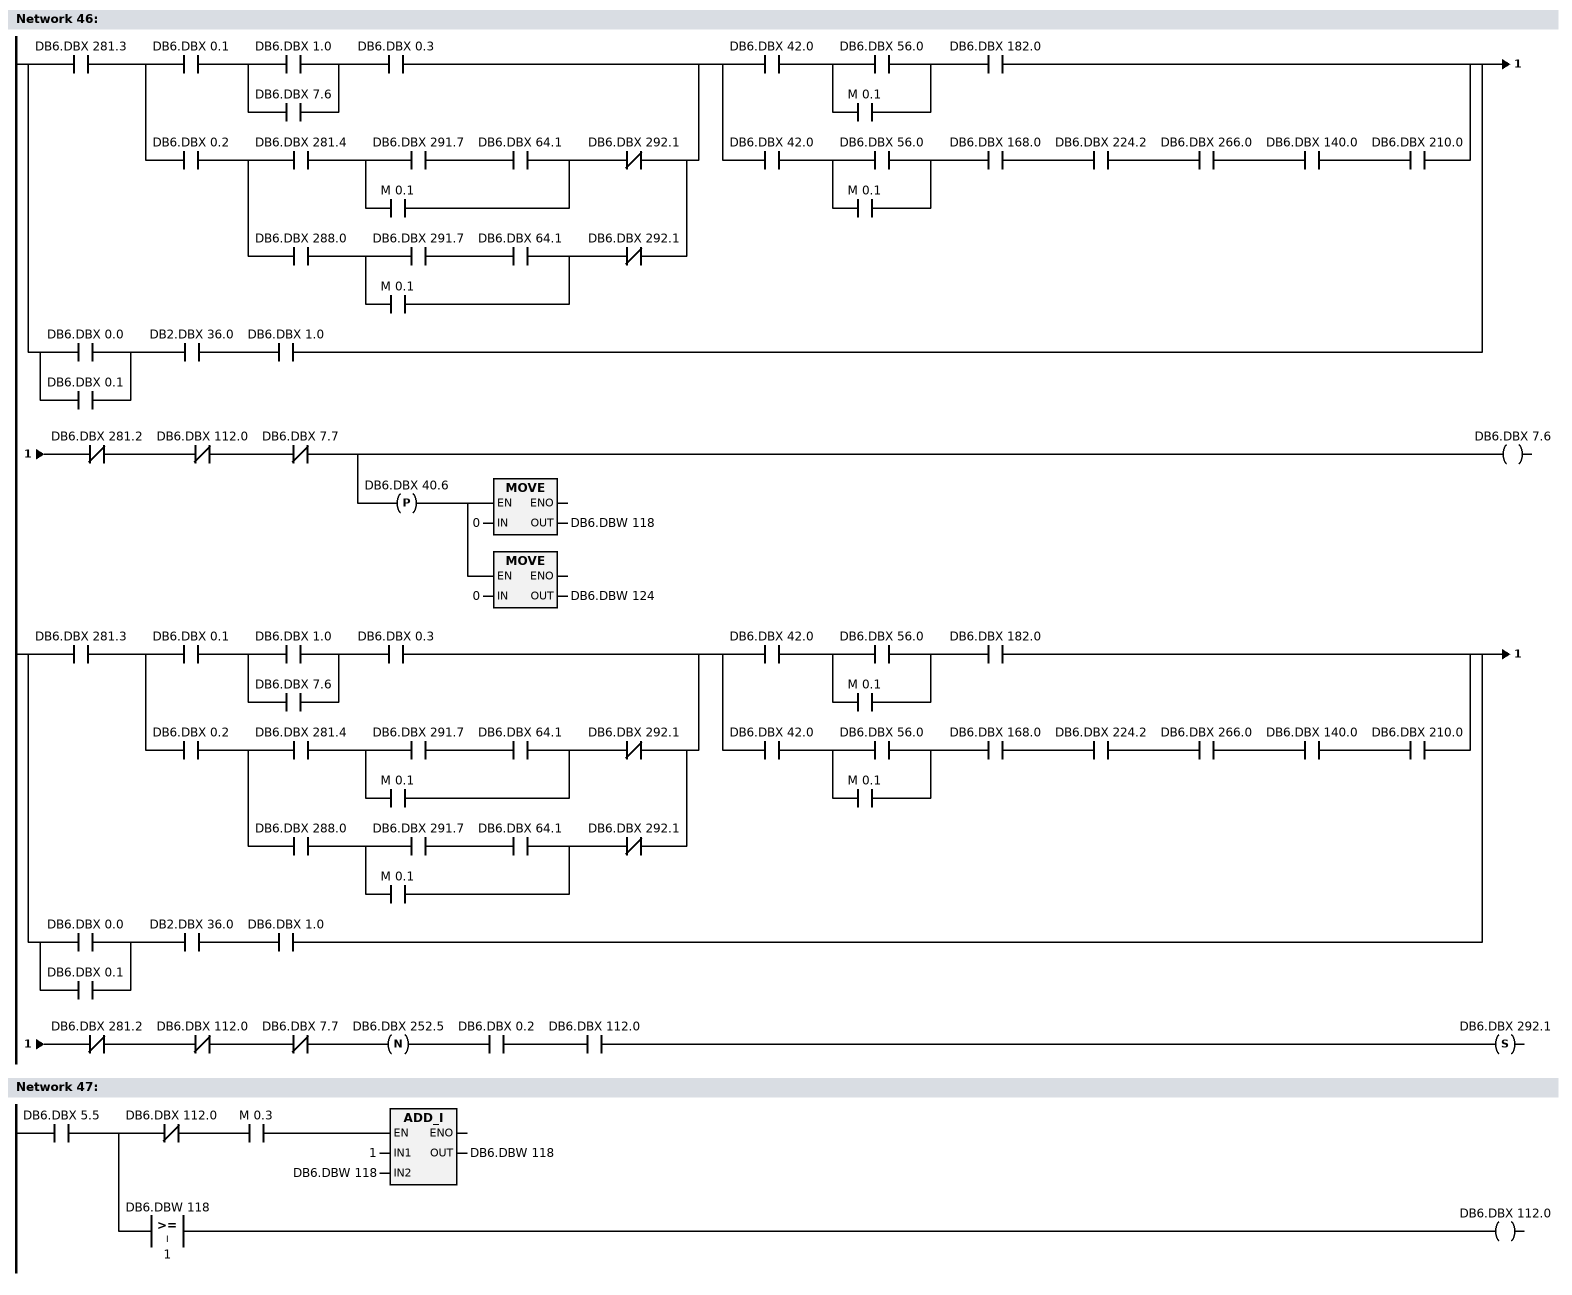
NETWORK
TITLE =
      A(;
      A     DB6.DBX 281.3;
      A(;
      A     DB6.DBX 0.1;
      A(;
      O     DB6.DBX 1.0;
      O     DB6.DBX 7.6;
      );
      A     DB6.DBX 0.3;
      O;
      A     DB6.DBX 0.2;
      A(;
      A     DB6.DBX 281.4;
      A(;
      A     DB6.DBX 291.7;
      A     DB6.DBX 64.1;
      O     M 0.1;
      );
      AN    DB6.DBX 292.1;
      O;
      A     DB6.DBX 288.0;
      A(;
      A     DB6.DBX 291.7;
      A     DB6.DBX 64.1;
      O     M 0.1;
      );
      AN    DB6.DBX 292.1;
      );
      );
      A(;
      A     DB6.DBX 42.0;
      A(;
      O     DB6.DBX 56.0;
      O     M 0.1;
      );
      A     DB6.DBX 182.0;
      O;
      A     DB6.DBX 42.0;
      A(;
      O     DB6.DBX 56.0;
      O     M 0.1;
      );
      A     DB6.DBX 168.0;
      A     DB6.DBX 224.2;
      A     DB6.DBX 266.0;
      A     DB6.DBX 140.0;
      A     DB6.DBX 210.0;
      );
      O;
      A(;
      O     DB6.DBX 0.0;
      O     DB6.DBX 0.1;
      );
      A     DB2.DBX 36.0;
      A     DB6.DBX 1.0;
      );
      AN    DB6.DBX 281.2;
      AN    DB6.DBX 112.0;
      AN    DB6.DBX 7.7;
      =     L 0.0;
      A     L 0.0;
      BLD   102;
      =     DB6.DBX 7.6;
      A(;
      A     L 0.0;
      FN    DB6.DBX 252.5;
      );
      A     DB6.DBX 0.2;
      A     DB6.DBX 112.0;
      S     DB6.DBX 292.1;
      A     L 0.0;
      FP    DB6.DBX 40.6;
      =     L 0.1;
      A     L 0.1;
      JNB   M039;
      L     0;
      T     DB6.DBW 118;
M039: NOP   0;
      A     L 0.1;
      JNB   M040;
      L     0;
      T     DB6.DBW 124;
M040: NOP   0;
NETWORK
TITLE =
      A     DB6.DBX 5.5;
      =     L 0.0;
      A     L 0.0;
      AN    DB6.DBX 112.0;
      A     M 0.3;
      JNB   M041;
      L     1;
      L     DB6.DBW 118;
      +I;
      T     DB6.DBW 118;
M041: NOP   0;
      A     L 0.0;
      A(;
      L     DB6.DBW 118;
      L     1;
      >=I;
      );
      =     DB6.DBX 112.0;
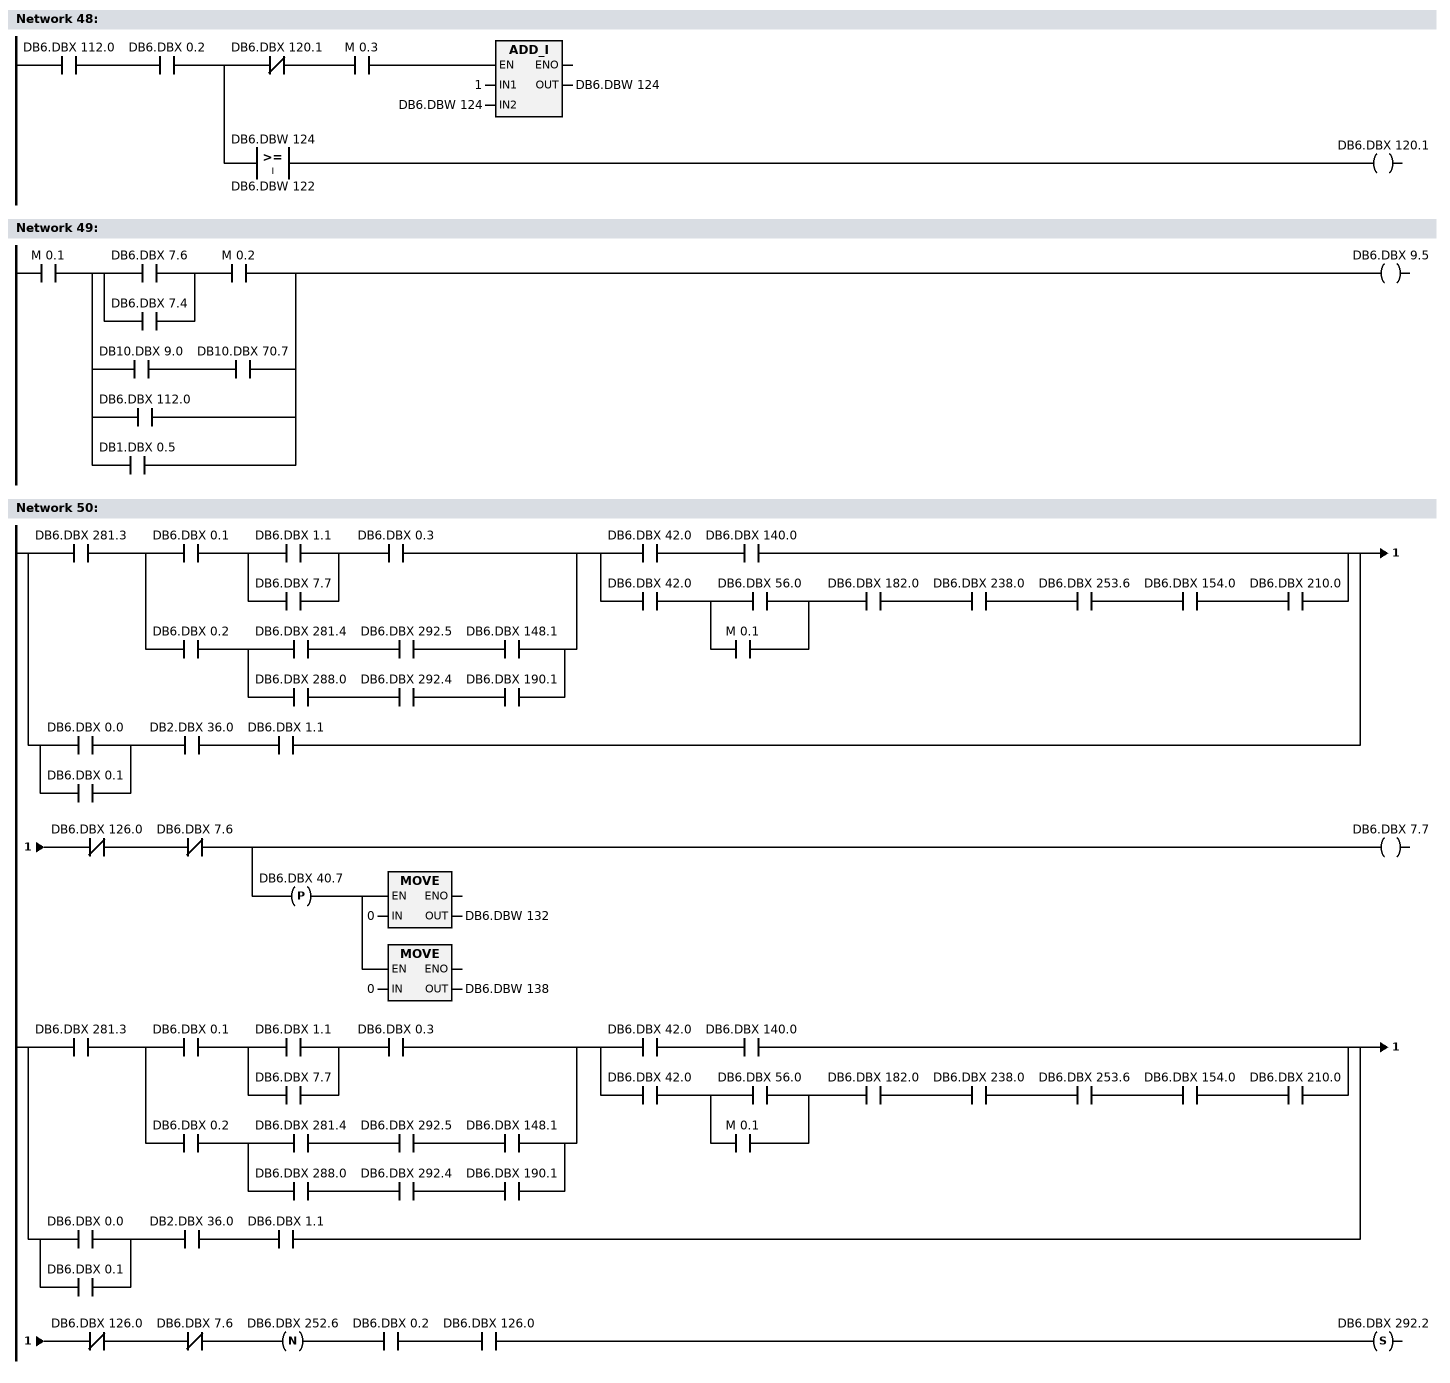
NETWORK
TITLE =
      A     DB6.DBX 112.0;
      A     DB6.DBX 0.2;
      =     L 0.0;
      A     L 0.0;
      AN    DB6.DBX 120.1;
      A     M 0.3;
      JNB   M042;
      L     1;
      L     DB6.DBW 124;
      +I;
      T     DB6.DBW 124;
M042: NOP   0;
      A     L 0.0;
      A(;
      L     DB6.DBW 124;
      L     DB6.DBW 122;
      >=I;
      );
      =     DB6.DBX 120.1;
NETWORK
TITLE =
      A     M 0.1;
      A(;
      A(;
      O     DB6.DBX 7.6;
      O     DB6.DBX 7.4;
      );
      A     M 0.2;
      O;
      A     DB10.DBX 9.0;
      A     DB10.DBX 70.7;
      O     DB6.DBX 112.0;
      O     DB1.DBX 0.5;
      );
      =     DB6.DBX 9.5;
NETWORK
TITLE =
      A(;
      A     DB6.DBX 281.3;
      A(;
      A     DB6.DBX 0.1;
      A(;
      O     DB6.DBX 1.1;
      O     DB6.DBX 7.7;
      );
      A     DB6.DBX 0.3;
      O;
      A     DB6.DBX 0.2;
      A(;
      A     DB6.DBX 281.4;
      A     DB6.DBX 292.5;
      A     DB6.DBX 148.1;
      O;
      A     DB6.DBX 288.0;
      A     DB6.DBX 292.4;
      A     DB6.DBX 190.1;
      );
      );
      A(;
      A     DB6.DBX 42.0;
      A     DB6.DBX 140.0;
      O;
      A     DB6.DBX 42.0;
      A(;
      O     DB6.DBX 56.0;
      O     M 0.1;
      );
      A     DB6.DBX 182.0;
      A     DB6.DBX 238.0;
      A     DB6.DBX 253.6;
      A     DB6.DBX 154.0;
      A     DB6.DBX 210.0;
      );
      O;
      A(;
      O     DB6.DBX 0.0;
      O     DB6.DBX 0.1;
      );
      A     DB2.DBX 36.0;
      A     DB6.DBX 1.1;
      );
      AN    DB6.DBX 126.0;
      AN    DB6.DBX 7.6;
      =     L 0.0;
      A     L 0.0;
      BLD   102;
      =     DB6.DBX 7.7;
      A(;
      A     L 0.0;
      FN    DB6.DBX 252.6;
      );
      A     DB6.DBX 0.2;
      A     DB6.DBX 126.0;
      S     DB6.DBX 292.2;
      A     L 0.0;
      FP    DB6.DBX 40.7;
      =     L 0.1;
      A     L 0.1;
      JNB   M043;
      L     0;
      T     DB6.DBW 132;
M043: NOP   0;
      A     L 0.1;
      JNB   M044;
      L     0;
      T     DB6.DBW 138;
M044: NOP   0;
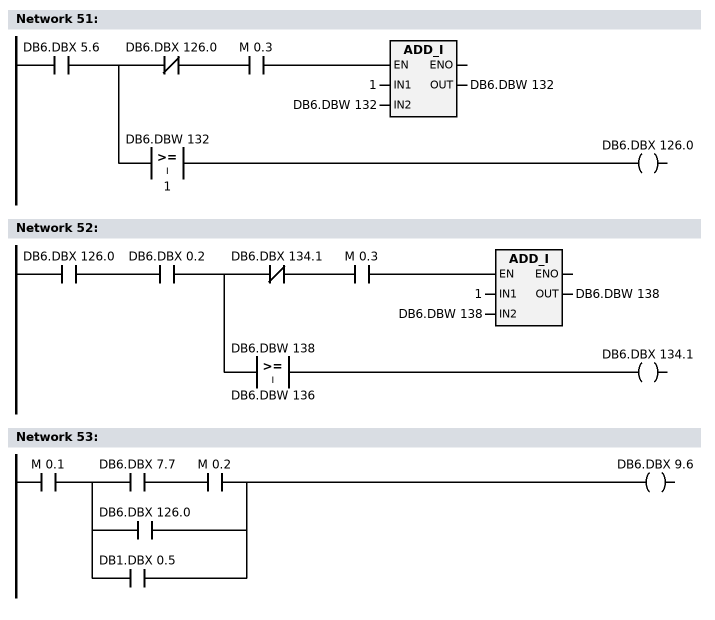
NETWORK
TITLE =
      A     DB6.DBX 5.6;
      =     L 0.0;
      A     L 0.0;
      AN    DB6.DBX 126.0;
      A     M 0.3;
      JNB   M045;
      L     1;
      L     DB6.DBW 132;
      +I;
      T     DB6.DBW 132;
M045: NOP   0;
      A     L 0.0;
      A(;
      L     DB6.DBW 132;
      L     1;
      >=I;
      );
      =     DB6.DBX 126.0;
NETWORK
TITLE =
      A     DB6.DBX 126.0;
      A     DB6.DBX 0.2;
      =     L 0.0;
      A     L 0.0;
      AN    DB6.DBX 134.1;
      A     M 0.3;
      JNB   M046;
      L     1;
      L     DB6.DBW 138;
      +I;
      T     DB6.DBW 138;
M046: NOP   0;
      A     L 0.0;
      A(;
      L     DB6.DBW 138;
      L     DB6.DBW 136;
      >=I;
      );
      =     DB6.DBX 134.1;
NETWORK
TITLE =
      A     M 0.1;
      A(;
      A     DB6.DBX 7.7;
      A     M 0.2;
      O     DB6.DBX 126.0;
      O     DB1.DBX 0.5;
      );
      =     DB6.DBX 9.6;
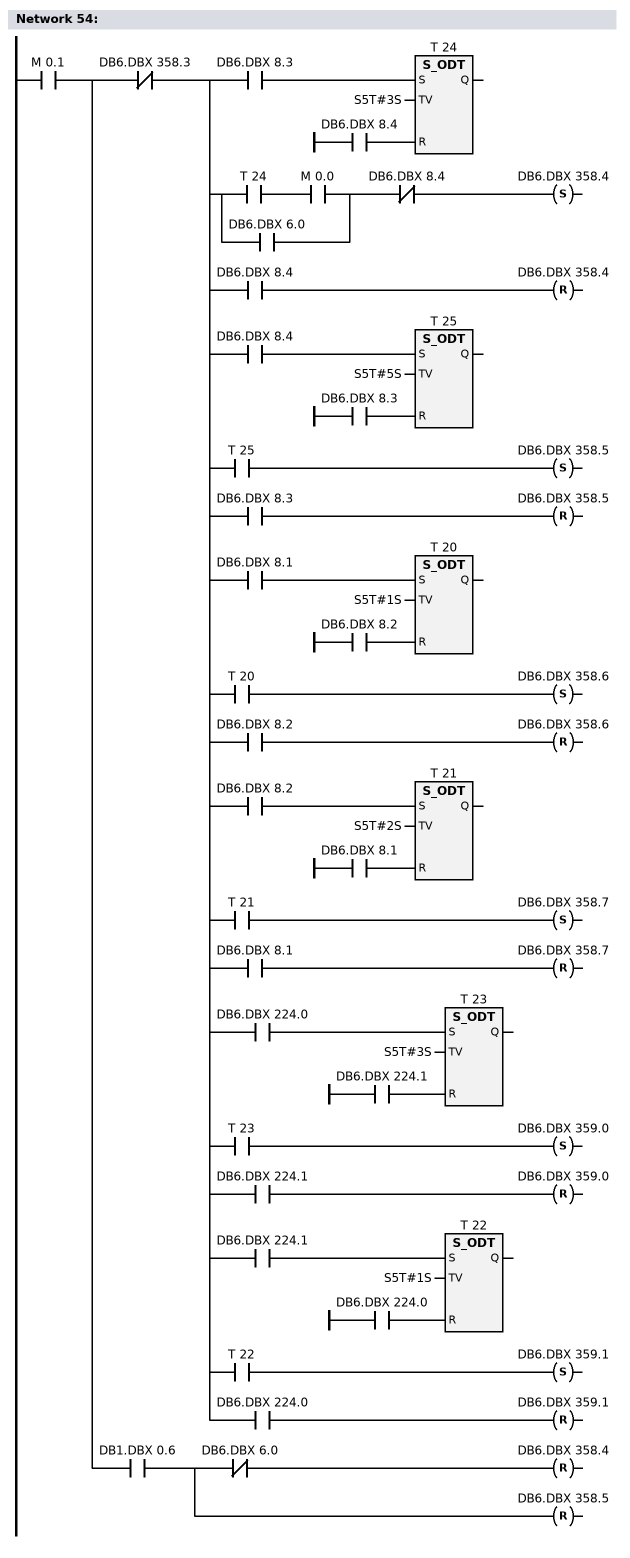
NETWORK
TITLE =
      A     M 0.1;
      =     L 0.0;
      A     L 0.0;
      AN    DB6.DBX 358.3;
      =     L 0.1;
      A     L 0.1;
      A     DB6.DBX 8.3;
      L     S5T#3S;
      SD    T 24;
      A     DB6.DBX 8.4;
      R     T 24;
      NOP   0;
      NOP   0;
      NOP   0;
      A     L 0.1;
      A(;
      A     T 24;
      A     M 0.0;
      O     DB6.DBX 6.0;
      );
      AN    DB6.DBX 8.4;
      S     DB6.DBX 358.4;
      A     L 0.1;
      A     DB6.DBX 8.4;
      R     DB6.DBX 358.4;
      A     L 0.1;
      A     DB6.DBX 8.4;
      L     S5T#5S;
      SD    T 25;
      A     DB6.DBX 8.3;
      R     T 25;
      NOP   0;
      NOP   0;
      NOP   0;
      A     L 0.1;
      A     T 25;
      S     DB6.DBX 358.5;
      A     L 0.1;
      A     DB6.DBX 8.3;
      R     DB6.DBX 358.5;
      A     L 0.1;
      A     DB6.DBX 8.1;
      L     S5T#1S;
      SD    T 20;
      A     DB6.DBX 8.2;
      R     T 20;
      NOP   0;
      NOP   0;
      NOP   0;
      A     L 0.1;
      A     T 20;
      S     DB6.DBX 358.6;
      A     L 0.1;
      A     DB6.DBX 8.2;
      R     DB6.DBX 358.6;
      A     L 0.1;
      A     DB6.DBX 8.2;
      L     S5T#2S;
      SD    T 21;
      A     DB6.DBX 8.1;
      R     T 21;
      NOP   0;
      NOP   0;
      NOP   0;
      A     L 0.1;
      A     T 21;
      S     DB6.DBX 358.7;
      A     L 0.1;
      A     DB6.DBX 8.1;
      R     DB6.DBX 358.7;
      A     L 0.1;
      A     DB6.DBX 224.0;
      L     S5T#3S;
      SD    T 23;
      A     DB6.DBX 224.1;
      R     T 23;
      NOP   0;
      NOP   0;
      NOP   0;
      A     L 0.1;
      A     T 23;
      S     DB6.DBX 359.0;
      A     L 0.1;
      A     DB6.DBX 224.1;
      R     DB6.DBX 359.0;
      A     L 0.1;
      A     DB6.DBX 224.1;
      L     S5T#1S;
      SD    T 22;
      A     DB6.DBX 224.0;
      R     T 22;
      NOP   0;
      NOP   0;
      NOP   0;
      A     L 0.1;
      A     T 22;
      S     DB6.DBX 359.1;
      A     L 0.1;
      A     DB6.DBX 224.0;
      R     DB6.DBX 359.1;
      A     L 0.0;
      A     DB1.DBX 0.6;
      =     L 0.1;
      A     L 0.1;
      AN    DB6.DBX 6.0;
      R     DB6.DBX 358.4;
      A     L 0.1;
      BLD   102;
      R     DB6.DBX 358.5;
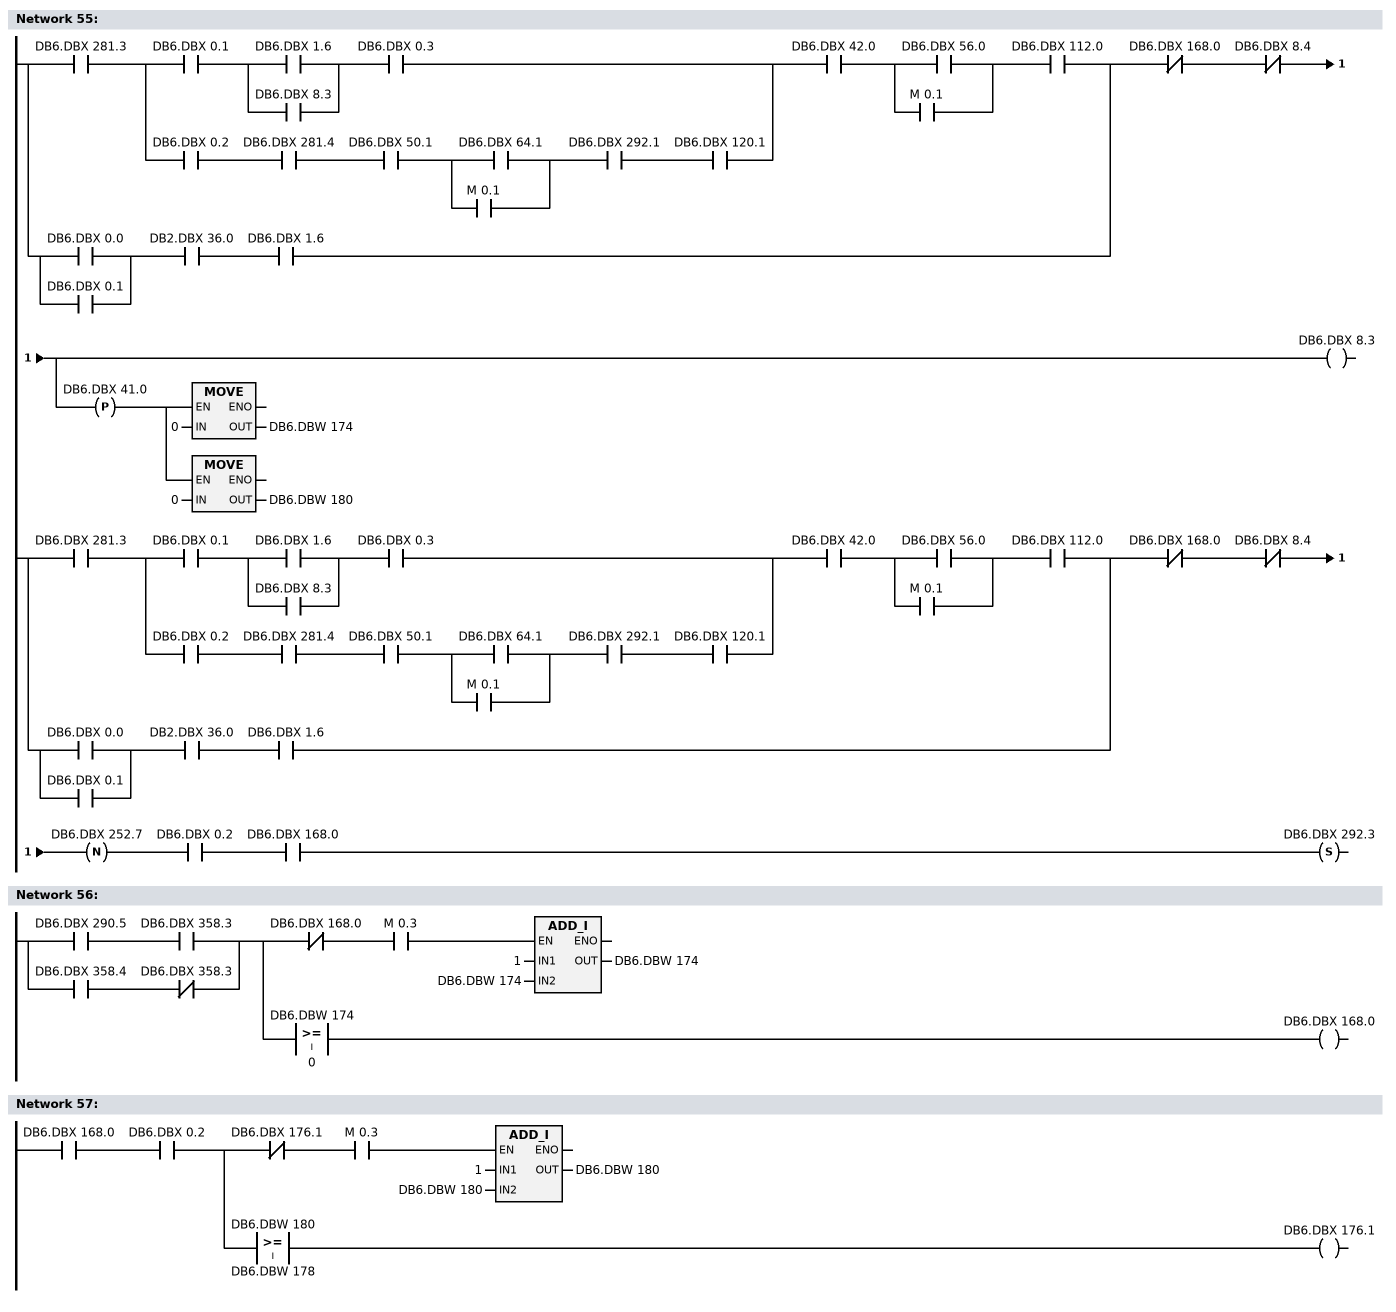
NETWORK
TITLE =
      A(;
      A     DB6.DBX 281.3;
      A(;
      A     DB6.DBX 0.1;
      A(;
      O     DB6.DBX 1.6;
      O     DB6.DBX 8.3;
      );
      A     DB6.DBX 0.3;
      O;
      A     DB6.DBX 0.2;
      A     DB6.DBX 281.4;
      A     DB6.DBX 50.1;
      A(;
      O     DB6.DBX 64.1;
      O     M 0.1;
      );
      A     DB6.DBX 292.1;
      A     DB6.DBX 120.1;
      );
      A     DB6.DBX 42.0;
      A(;
      O     DB6.DBX 56.0;
      O     M 0.1;
      );
      A     DB6.DBX 112.0;
      O;
      A(;
      O     DB6.DBX 0.0;
      O     DB6.DBX 0.1;
      );
      A     DB2.DBX 36.0;
      A     DB6.DBX 1.6;
      );
      AN    DB6.DBX 168.0;
      AN    DB6.DBX 8.4;
      =     L 0.0;
      A     L 0.0;
      BLD   102;
      =     DB6.DBX 8.3;
      A(;
      A     L 0.0;
      FN    DB6.DBX 252.7;
      );
      A     DB6.DBX 0.2;
      A     DB6.DBX 168.0;
      S     DB6.DBX 292.3;
      A     L 0.0;
      FP    DB6.DBX 41.0;
      =     L 0.1;
      A     L 0.1;
      JNB   M047;
      L     0;
      T     DB6.DBW 174;
M047: NOP   0;
      A     L 0.1;
      JNB   M048;
      L     0;
      T     DB6.DBW 180;
M048: NOP   0;
NETWORK
TITLE =
      A     DB6.DBX 290.5;
      A     DB6.DBX 358.3;
      O;
      A     DB6.DBX 358.4;
      AN    DB6.DBX 358.3;
      =     L 0.0;
      A     L 0.0;
      AN    DB6.DBX 168.0;
      A     M 0.3;
      JNB   M049;
      L     1;
      L     DB6.DBW 174;
      +I;
      T     DB6.DBW 174;
M049: NOP   0;
      A     L 0.0;
      A(;
      L     DB6.DBW 174;
      L     0;
      >=I;
      );
      =     DB6.DBX 168.0;
NETWORK
TITLE =
      A     DB6.DBX 168.0;
      A     DB6.DBX 0.2;
      =     L 0.0;
      A     L 0.0;
      AN    DB6.DBX 176.1;
      A     M 0.3;
      JNB   M050;
      L     1;
      L     DB6.DBW 180;
      +I;
      T     DB6.DBW 180;
M050: NOP   0;
      A     L 0.0;
      A(;
      L     DB6.DBW 180;
      L     DB6.DBW 178;
      >=I;
      );
      =     DB6.DBX 176.1;
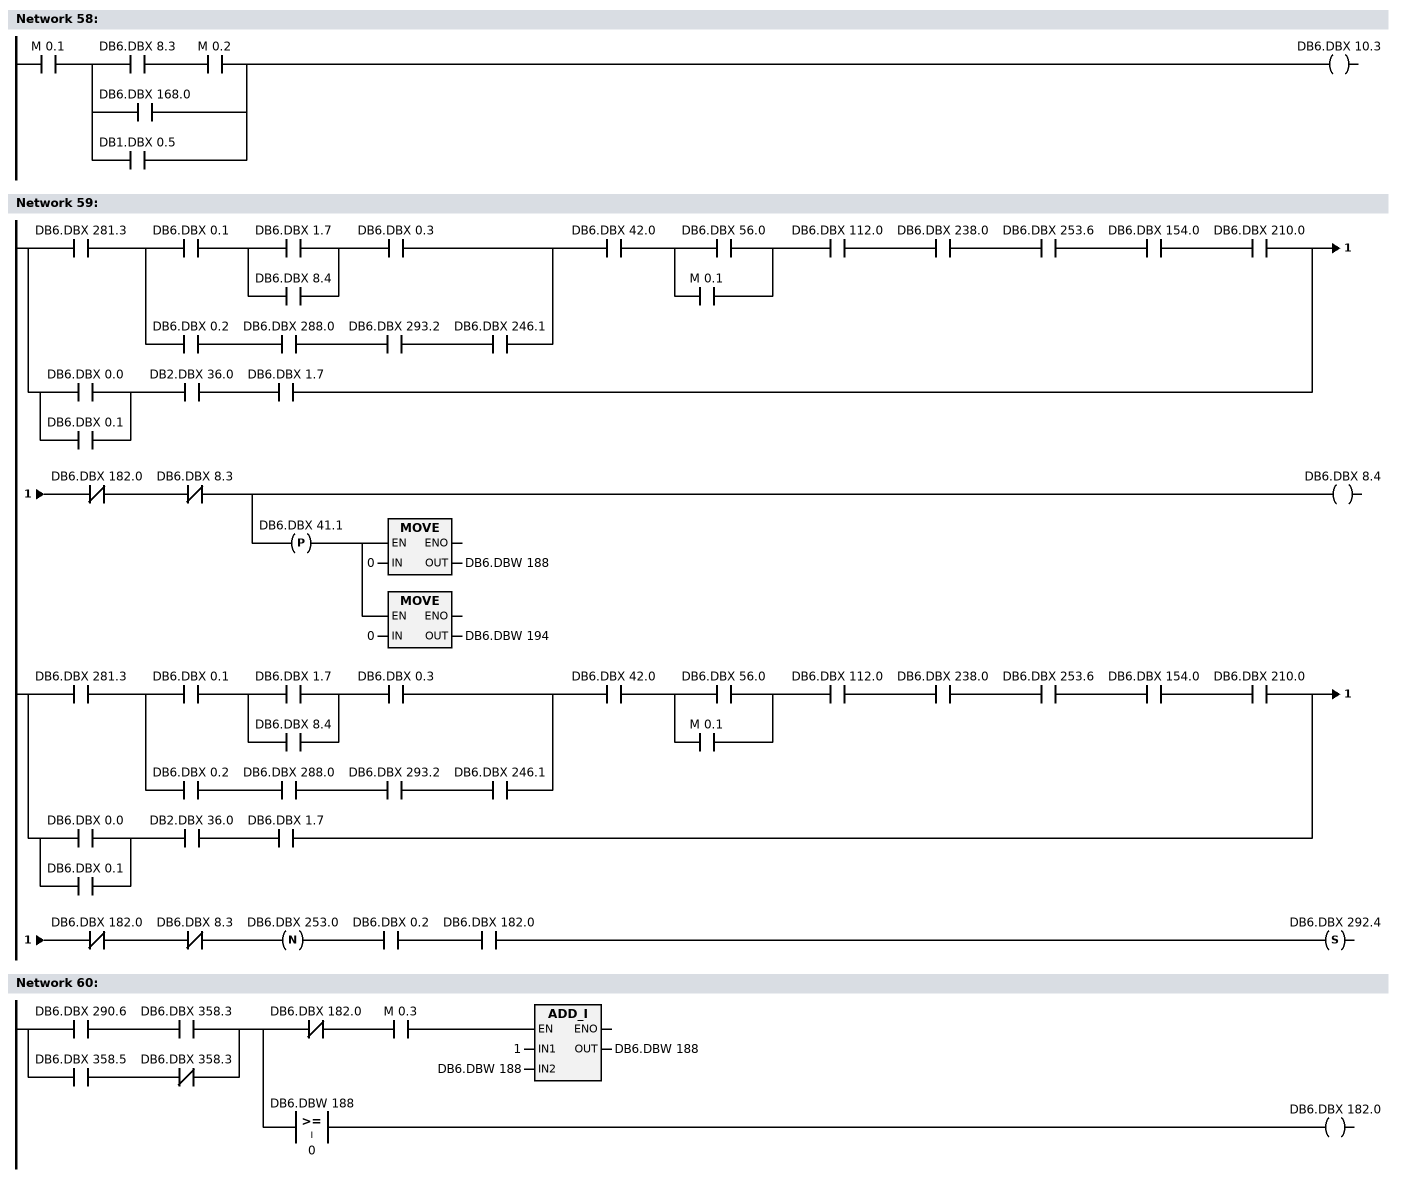
NETWORK
TITLE =
      A     M 0.1;
      A(;
      A     DB6.DBX 8.3;
      A     M 0.2;
      O     DB6.DBX 168.0;
      O     DB1.DBX 0.5;
      );
      =     DB6.DBX 10.3;
NETWORK
TITLE =
      A(;
      A     DB6.DBX 281.3;
      A(;
      A     DB6.DBX 0.1;
      A(;
      O     DB6.DBX 1.7;
      O     DB6.DBX 8.4;
      );
      A     DB6.DBX 0.3;
      O;
      A     DB6.DBX 0.2;
      A     DB6.DBX 288.0;
      A     DB6.DBX 293.2;
      A     DB6.DBX 246.1;
      );
      A     DB6.DBX 42.0;
      A(;
      O     DB6.DBX 56.0;
      O     M 0.1;
      );
      A     DB6.DBX 112.0;
      A     DB6.DBX 238.0;
      A     DB6.DBX 253.6;
      A     DB6.DBX 154.0;
      A     DB6.DBX 210.0;
      O;
      A(;
      O     DB6.DBX 0.0;
      O     DB6.DBX 0.1;
      );
      A     DB2.DBX 36.0;
      A     DB6.DBX 1.7;
      );
      AN    DB6.DBX 182.0;
      AN    DB6.DBX 8.3;
      =     L 0.0;
      A     L 0.0;
      BLD   102;
      =     DB6.DBX 8.4;
      A(;
      A     L 0.0;
      FN    DB6.DBX 253.0;
      );
      A     DB6.DBX 0.2;
      A     DB6.DBX 182.0;
      S     DB6.DBX 292.4;
      A     L 0.0;
      FP    DB6.DBX 41.1;
      =     L 0.1;
      A     L 0.1;
      JNB   M051;
      L     0;
      T     DB6.DBW 188;
M051: NOP   0;
      A     L 0.1;
      JNB   M052;
      L     0;
      T     DB6.DBW 194;
M052: NOP   0;
NETWORK
TITLE =
      A     DB6.DBX 290.6;
      A     DB6.DBX 358.3;
      O;
      A     DB6.DBX 358.5;
      AN    DB6.DBX 358.3;
      =     L 0.0;
      A     L 0.0;
      AN    DB6.DBX 182.0;
      A     M 0.3;
      JNB   M053;
      L     1;
      L     DB6.DBW 188;
      +I;
      T     DB6.DBW 188;
M053: NOP   0;
      A     L 0.0;
      A(;
      L     DB6.DBW 188;
      L     0;
      >=I;
      );
      =     DB6.DBX 182.0;
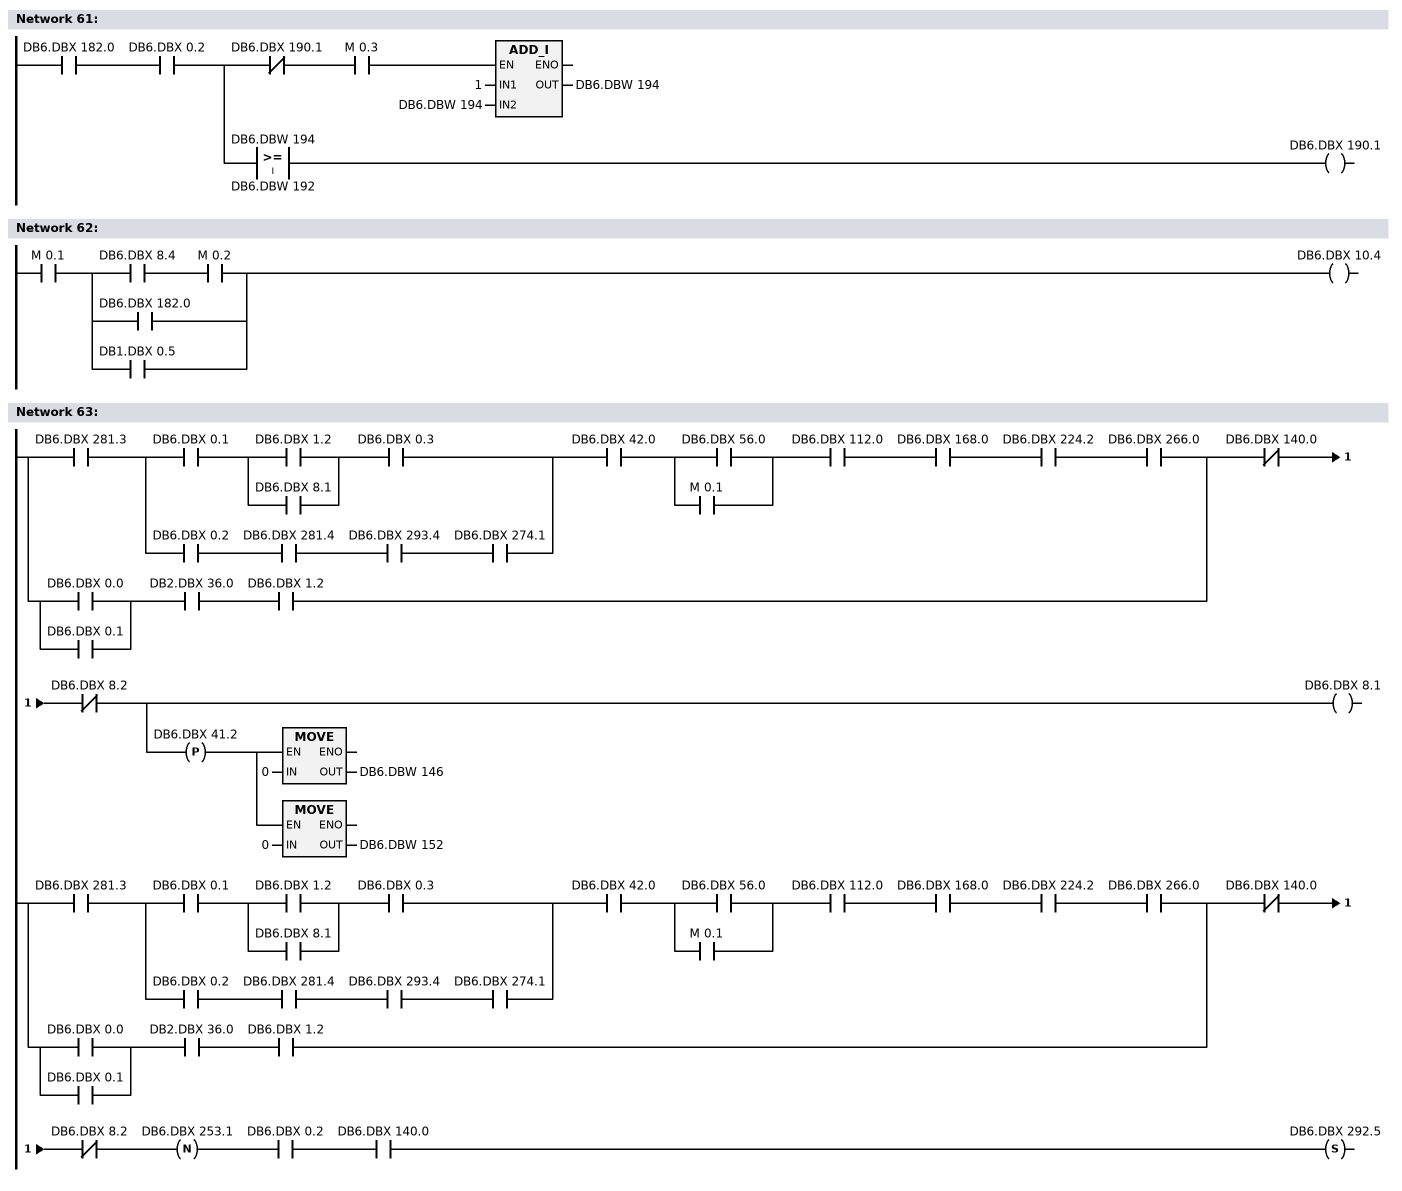
NETWORK
TITLE =
      A     DB6.DBX 182.0;
      A     DB6.DBX 0.2;
      =     L 0.0;
      A     L 0.0;
      AN    DB6.DBX 190.1;
      A     M 0.3;
      JNB   M054;
      L     1;
      L     DB6.DBW 194;
      +I;
      T     DB6.DBW 194;
M054: NOP   0;
      A     L 0.0;
      A(;
      L     DB6.DBW 194;
      L     DB6.DBW 192;
      >=I;
      );
      =     DB6.DBX 190.1;
NETWORK
TITLE =
      A     M 0.1;
      A(;
      A     DB6.DBX 8.4;
      A     M 0.2;
      O     DB6.DBX 182.0;
      O     DB1.DBX 0.5;
      );
      =     DB6.DBX 10.4;
NETWORK
TITLE =
      A(;
      A     DB6.DBX 281.3;
      A(;
      A     DB6.DBX 0.1;
      A(;
      O     DB6.DBX 1.2;
      O     DB6.DBX 8.1;
      );
      A     DB6.DBX 0.3;
      O;
      A     DB6.DBX 0.2;
      A     DB6.DBX 281.4;
      A     DB6.DBX 293.4;
      A     DB6.DBX 274.1;
      );
      A     DB6.DBX 42.0;
      A(;
      O     DB6.DBX 56.0;
      O     M 0.1;
      );
      A     DB6.DBX 112.0;
      A     DB6.DBX 168.0;
      A     DB6.DBX 224.2;
      A     DB6.DBX 266.0;
      O;
      A(;
      O     DB6.DBX 0.0;
      O     DB6.DBX 0.1;
      );
      A     DB2.DBX 36.0;
      A     DB6.DBX 1.2;
      );
      AN    DB6.DBX 140.0;
      AN    DB6.DBX 8.2;
      =     L 0.0;
      A     L 0.0;
      BLD   102;
      =     DB6.DBX 8.1;
      A(;
      A     L 0.0;
      FN    DB6.DBX 253.1;
      );
      A     DB6.DBX 0.2;
      A     DB6.DBX 140.0;
      S     DB6.DBX 292.5;
      A     L 0.0;
      FP    DB6.DBX 41.2;
      =     L 0.1;
      A     L 0.1;
      JNB   M055;
      L     0;
      T     DB6.DBW 146;
M055: NOP   0;
      A     L 0.1;
      JNB   M056;
      L     0;
      T     DB6.DBW 152;
M056: NOP   0;
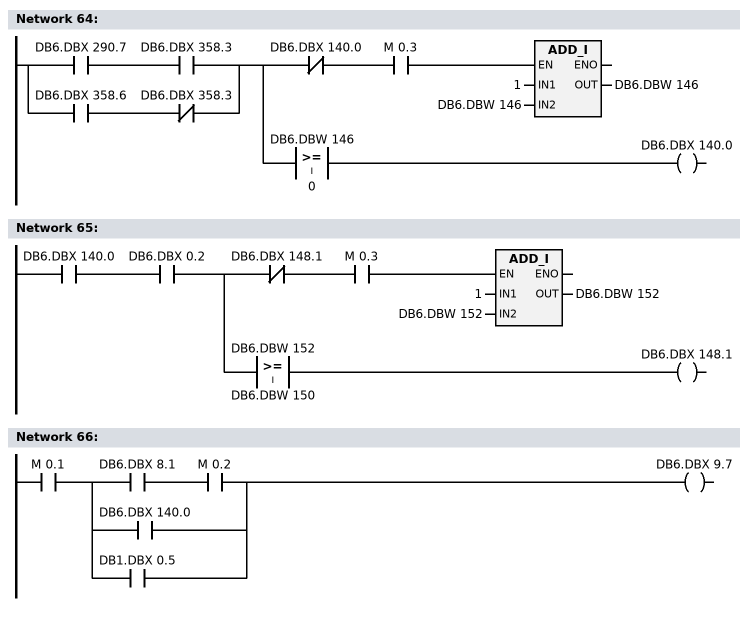
NETWORK
TITLE =
      A     DB6.DBX 290.7;
      A     DB6.DBX 358.3;
      O;
      A     DB6.DBX 358.6;
      AN    DB6.DBX 358.3;
      =     L 0.0;
      A     L 0.0;
      AN    DB6.DBX 140.0;
      A     M 0.3;
      JNB   M057;
      L     1;
      L     DB6.DBW 146;
      +I;
      T     DB6.DBW 146;
M057: NOP   0;
      A     L 0.0;
      A(;
      L     DB6.DBW 146;
      L     0;
      >=I;
      );
      =     DB6.DBX 140.0;
NETWORK
TITLE =
      A     DB6.DBX 140.0;
      A     DB6.DBX 0.2;
      =     L 0.0;
      A     L 0.0;
      AN    DB6.DBX 148.1;
      A     M 0.3;
      JNB   M058;
      L     1;
      L     DB6.DBW 152;
      +I;
      T     DB6.DBW 152;
M058: NOP   0;
      A     L 0.0;
      A(;
      L     DB6.DBW 152;
      L     DB6.DBW 150;
      >=I;
      );
      =     DB6.DBX 148.1;
NETWORK
TITLE =
      A     M 0.1;
      A(;
      A     DB6.DBX 8.1;
      A     M 0.2;
      O     DB6.DBX 140.0;
      O     DB1.DBX 0.5;
      );
      =     DB6.DBX 9.7;
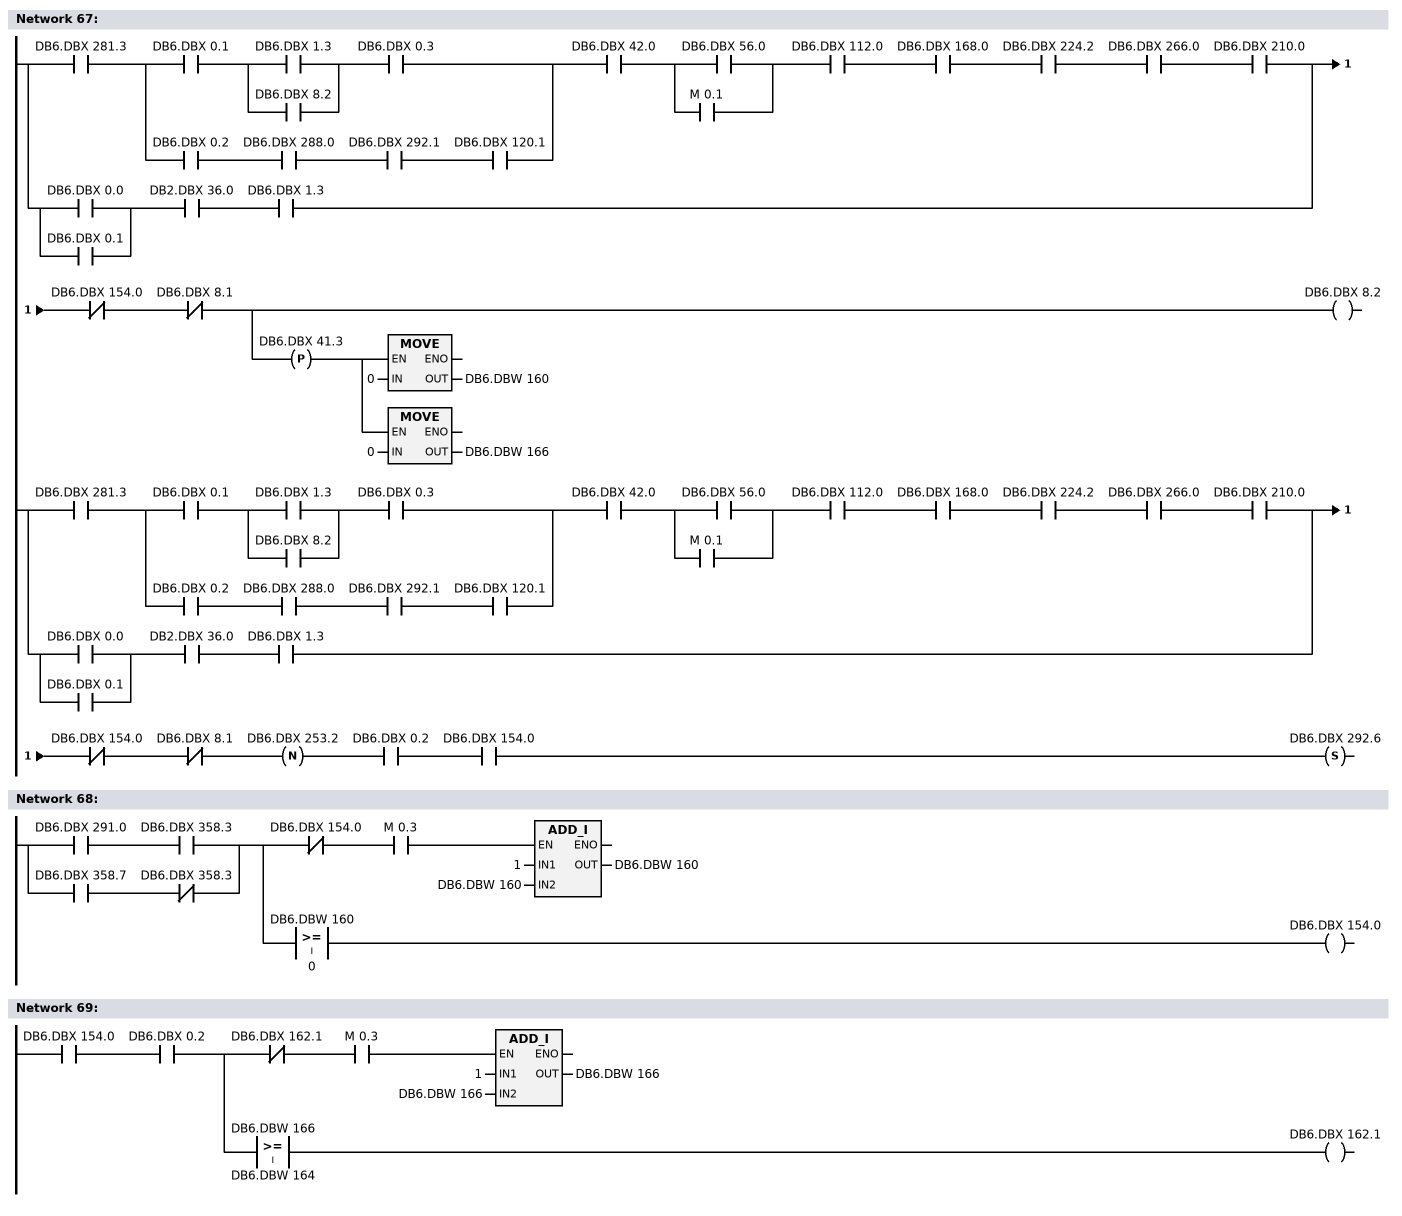
NETWORK
TITLE =
      A(;
      A     DB6.DBX 281.3;
      A(;
      A     DB6.DBX 0.1;
      A(;
      O     DB6.DBX 1.3;
      O     DB6.DBX 8.2;
      );
      A     DB6.DBX 0.3;
      O;
      A     DB6.DBX 0.2;
      A     DB6.DBX 288.0;
      A     DB6.DBX 292.1;
      A     DB6.DBX 120.1;
      );
      A     DB6.DBX 42.0;
      A(;
      O     DB6.DBX 56.0;
      O     M 0.1;
      );
      A     DB6.DBX 112.0;
      A     DB6.DBX 168.0;
      A     DB6.DBX 224.2;
      A     DB6.DBX 266.0;
      A     DB6.DBX 210.0;
      O;
      A(;
      O     DB6.DBX 0.0;
      O     DB6.DBX 0.1;
      );
      A     DB2.DBX 36.0;
      A     DB6.DBX 1.3;
      );
      AN    DB6.DBX 154.0;
      AN    DB6.DBX 8.1;
      =     L 0.0;
      A     L 0.0;
      BLD   102;
      =     DB6.DBX 8.2;
      A(;
      A     L 0.0;
      FN    DB6.DBX 253.2;
      );
      A     DB6.DBX 0.2;
      A     DB6.DBX 154.0;
      S     DB6.DBX 292.6;
      A     L 0.0;
      FP    DB6.DBX 41.3;
      =     L 0.1;
      A     L 0.1;
      JNB   M059;
      L     0;
      T     DB6.DBW 160;
M059: NOP   0;
      A     L 0.1;
      JNB   M060;
      L     0;
      T     DB6.DBW 166;
M060: NOP   0;
NETWORK
TITLE =
      A     DB6.DBX 291.0;
      A     DB6.DBX 358.3;
      O;
      A     DB6.DBX 358.7;
      AN    DB6.DBX 358.3;
      =     L 0.0;
      A     L 0.0;
      AN    DB6.DBX 154.0;
      A     M 0.3;
      JNB   M061;
      L     1;
      L     DB6.DBW 160;
      +I;
      T     DB6.DBW 160;
M061: NOP   0;
      A     L 0.0;
      A(;
      L     DB6.DBW 160;
      L     0;
      >=I;
      );
      =     DB6.DBX 154.0;
NETWORK
TITLE =
      A     DB6.DBX 154.0;
      A     DB6.DBX 0.2;
      =     L 0.0;
      A     L 0.0;
      AN    DB6.DBX 162.1;
      A     M 0.3;
      JNB   M062;
      L     1;
      L     DB6.DBW 166;
      +I;
      T     DB6.DBW 166;
M062: NOP   0;
      A     L 0.0;
      A(;
      L     DB6.DBW 166;
      L     DB6.DBW 164;
      >=I;
      );
      =     DB6.DBX 162.1;
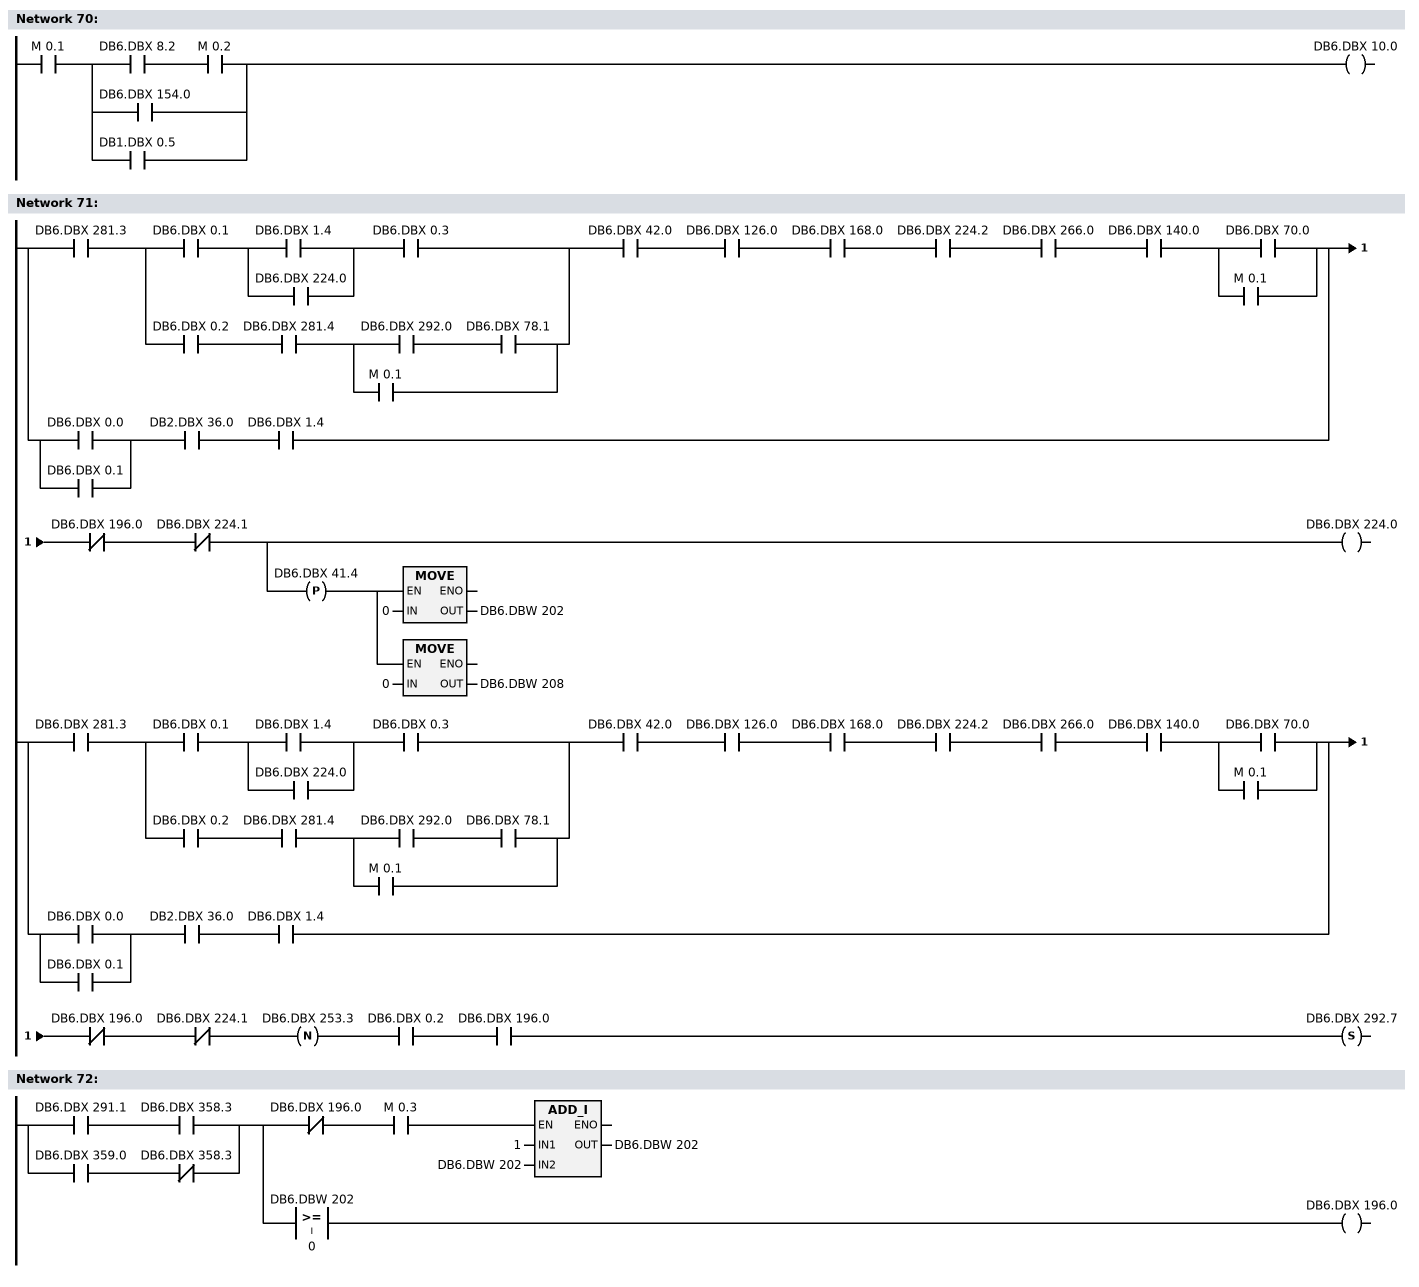
NETWORK
TITLE =
      A     M 0.1;
      A(;
      A     DB6.DBX 8.2;
      A     M 0.2;
      O     DB6.DBX 154.0;
      O     DB1.DBX 0.5;
      );
      =     DB6.DBX 10.0;
NETWORK
TITLE =
      A(;
      A     DB6.DBX 281.3;
      A(;
      A     DB6.DBX 0.1;
      A(;
      O     DB6.DBX 1.4;
      O     DB6.DBX 224.0;
      );
      A     DB6.DBX 0.3;
      O;
      A     DB6.DBX 0.2;
      A     DB6.DBX 281.4;
      A(;
      A     DB6.DBX 292.0;
      A     DB6.DBX 78.1;
      O     M 0.1;
      );
      );
      A     DB6.DBX 42.0;
      A     DB6.DBX 126.0;
      A     DB6.DBX 168.0;
      A     DB6.DBX 224.2;
      A     DB6.DBX 266.0;
      A     DB6.DBX 140.0;
      A(;
      O     DB6.DBX 70.0;
      O     M 0.1;
      );
      O;
      A(;
      O     DB6.DBX 0.0;
      O     DB6.DBX 0.1;
      );
      A     DB2.DBX 36.0;
      A     DB6.DBX 1.4;
      );
      AN    DB6.DBX 196.0;
      AN    DB6.DBX 224.1;
      =     L 0.0;
      A     L 0.0;
      BLD   102;
      =     DB6.DBX 224.0;
      A(;
      A     L 0.0;
      FN    DB6.DBX 253.3;
      );
      A     DB6.DBX 0.2;
      A     DB6.DBX 196.0;
      S     DB6.DBX 292.7;
      A     L 0.0;
      FP    DB6.DBX 41.4;
      =     L 0.1;
      A     L 0.1;
      JNB   M063;
      L     0;
      T     DB6.DBW 202;
M063: NOP   0;
      A     L 0.1;
      JNB   M064;
      L     0;
      T     DB6.DBW 208;
M064: NOP   0;
NETWORK
TITLE =
      A     DB6.DBX 291.1;
      A     DB6.DBX 358.3;
      O;
      A     DB6.DBX 359.0;
      AN    DB6.DBX 358.3;
      =     L 0.0;
      A     L 0.0;
      AN    DB6.DBX 196.0;
      A     M 0.3;
      JNB   M065;
      L     1;
      L     DB6.DBW 202;
      +I;
      T     DB6.DBW 202;
M065: NOP   0;
      A     L 0.0;
      A(;
      L     DB6.DBW 202;
      L     0;
      >=I;
      );
      =     DB6.DBX 196.0;
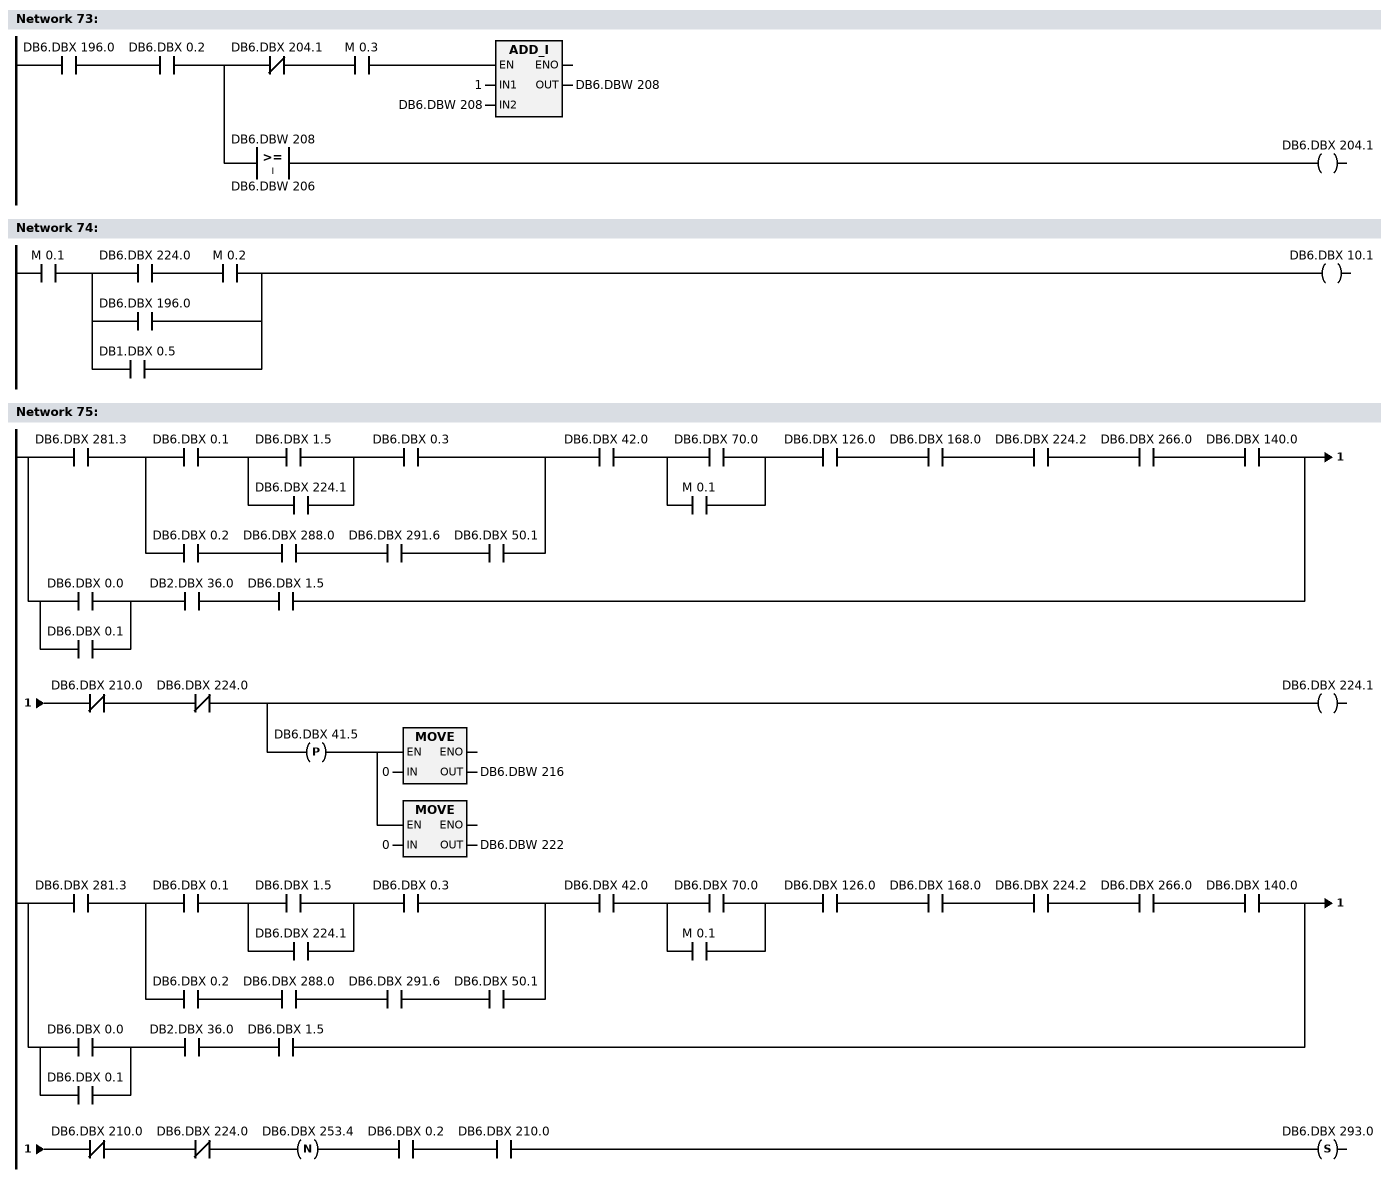
NETWORK
TITLE =
      A     DB6.DBX 196.0;
      A     DB6.DBX 0.2;
      =     L 0.0;
      A     L 0.0;
      AN    DB6.DBX 204.1;
      A     M 0.3;
      JNB   M066;
      L     1;
      L     DB6.DBW 208;
      +I;
      T     DB6.DBW 208;
M066: NOP   0;
      A     L 0.0;
      A(;
      L     DB6.DBW 208;
      L     DB6.DBW 206;
      >=I;
      );
      =     DB6.DBX 204.1;
NETWORK
TITLE =
      A     M 0.1;
      A(;
      A     DB6.DBX 224.0;
      A     M 0.2;
      O     DB6.DBX 196.0;
      O     DB1.DBX 0.5;
      );
      =     DB6.DBX 10.1;
NETWORK
TITLE =
      A(;
      A     DB6.DBX 281.3;
      A(;
      A     DB6.DBX 0.1;
      A(;
      O     DB6.DBX 1.5;
      O     DB6.DBX 224.1;
      );
      A     DB6.DBX 0.3;
      O;
      A     DB6.DBX 0.2;
      A     DB6.DBX 288.0;
      A     DB6.DBX 291.6;
      A     DB6.DBX 50.1;
      );
      A     DB6.DBX 42.0;
      A(;
      O     DB6.DBX 70.0;
      O     M 0.1;
      );
      A     DB6.DBX 126.0;
      A     DB6.DBX 168.0;
      A     DB6.DBX 224.2;
      A     DB6.DBX 266.0;
      A     DB6.DBX 140.0;
      O;
      A(;
      O     DB6.DBX 0.0;
      O     DB6.DBX 0.1;
      );
      A     DB2.DBX 36.0;
      A     DB6.DBX 1.5;
      );
      AN    DB6.DBX 210.0;
      AN    DB6.DBX 224.0;
      =     L 0.0;
      A     L 0.0;
      BLD   102;
      =     DB6.DBX 224.1;
      A(;
      A     L 0.0;
      FN    DB6.DBX 253.4;
      );
      A     DB6.DBX 0.2;
      A     DB6.DBX 210.0;
      S     DB6.DBX 293.0;
      A     L 0.0;
      FP    DB6.DBX 41.5;
      =     L 0.1;
      A     L 0.1;
      JNB   M067;
      L     0;
      T     DB6.DBW 216;
M067: NOP   0;
      A     L 0.1;
      JNB   M068;
      L     0;
      T     DB6.DBW 222;
M068: NOP   0;
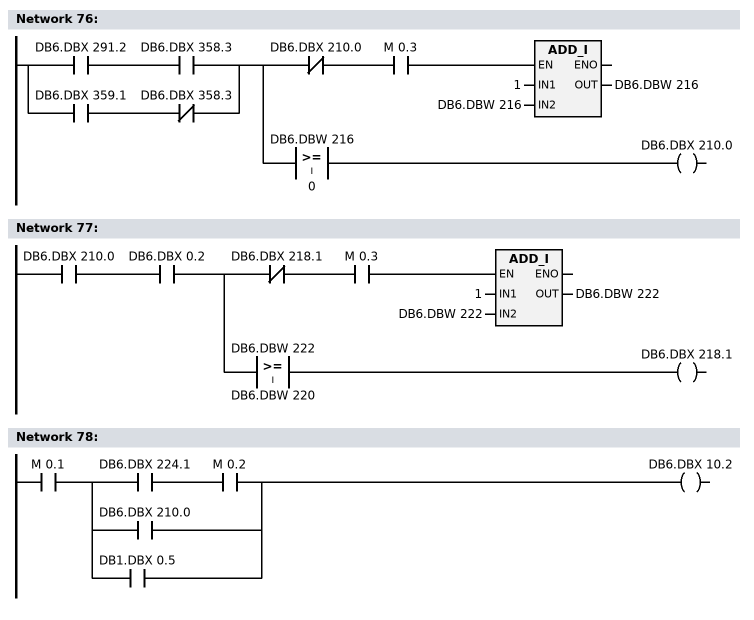
NETWORK
TITLE =
      A     DB6.DBX 291.2;
      A     DB6.DBX 358.3;
      O;
      A     DB6.DBX 359.1;
      AN    DB6.DBX 358.3;
      =     L 0.0;
      A     L 0.0;
      AN    DB6.DBX 210.0;
      A     M 0.3;
      JNB   M069;
      L     1;
      L     DB6.DBW 216;
      +I;
      T     DB6.DBW 216;
M069: NOP   0;
      A     L 0.0;
      A(;
      L     DB6.DBW 216;
      L     0;
      >=I;
      );
      =     DB6.DBX 210.0;
NETWORK
TITLE =
      A     DB6.DBX 210.0;
      A     DB6.DBX 0.2;
      =     L 0.0;
      A     L 0.0;
      AN    DB6.DBX 218.1;
      A     M 0.3;
      JNB   M070;
      L     1;
      L     DB6.DBW 222;
      +I;
      T     DB6.DBW 222;
M070: NOP   0;
      A     L 0.0;
      A(;
      L     DB6.DBW 222;
      L     DB6.DBW 220;
      >=I;
      );
      =     DB6.DBX 218.1;
NETWORK
TITLE =
      A     M 0.1;
      A(;
      A     DB6.DBX 224.1;
      A     M 0.2;
      O     DB6.DBX 210.0;
      O     DB1.DBX 0.5;
      );
      =     DB6.DBX 10.2;
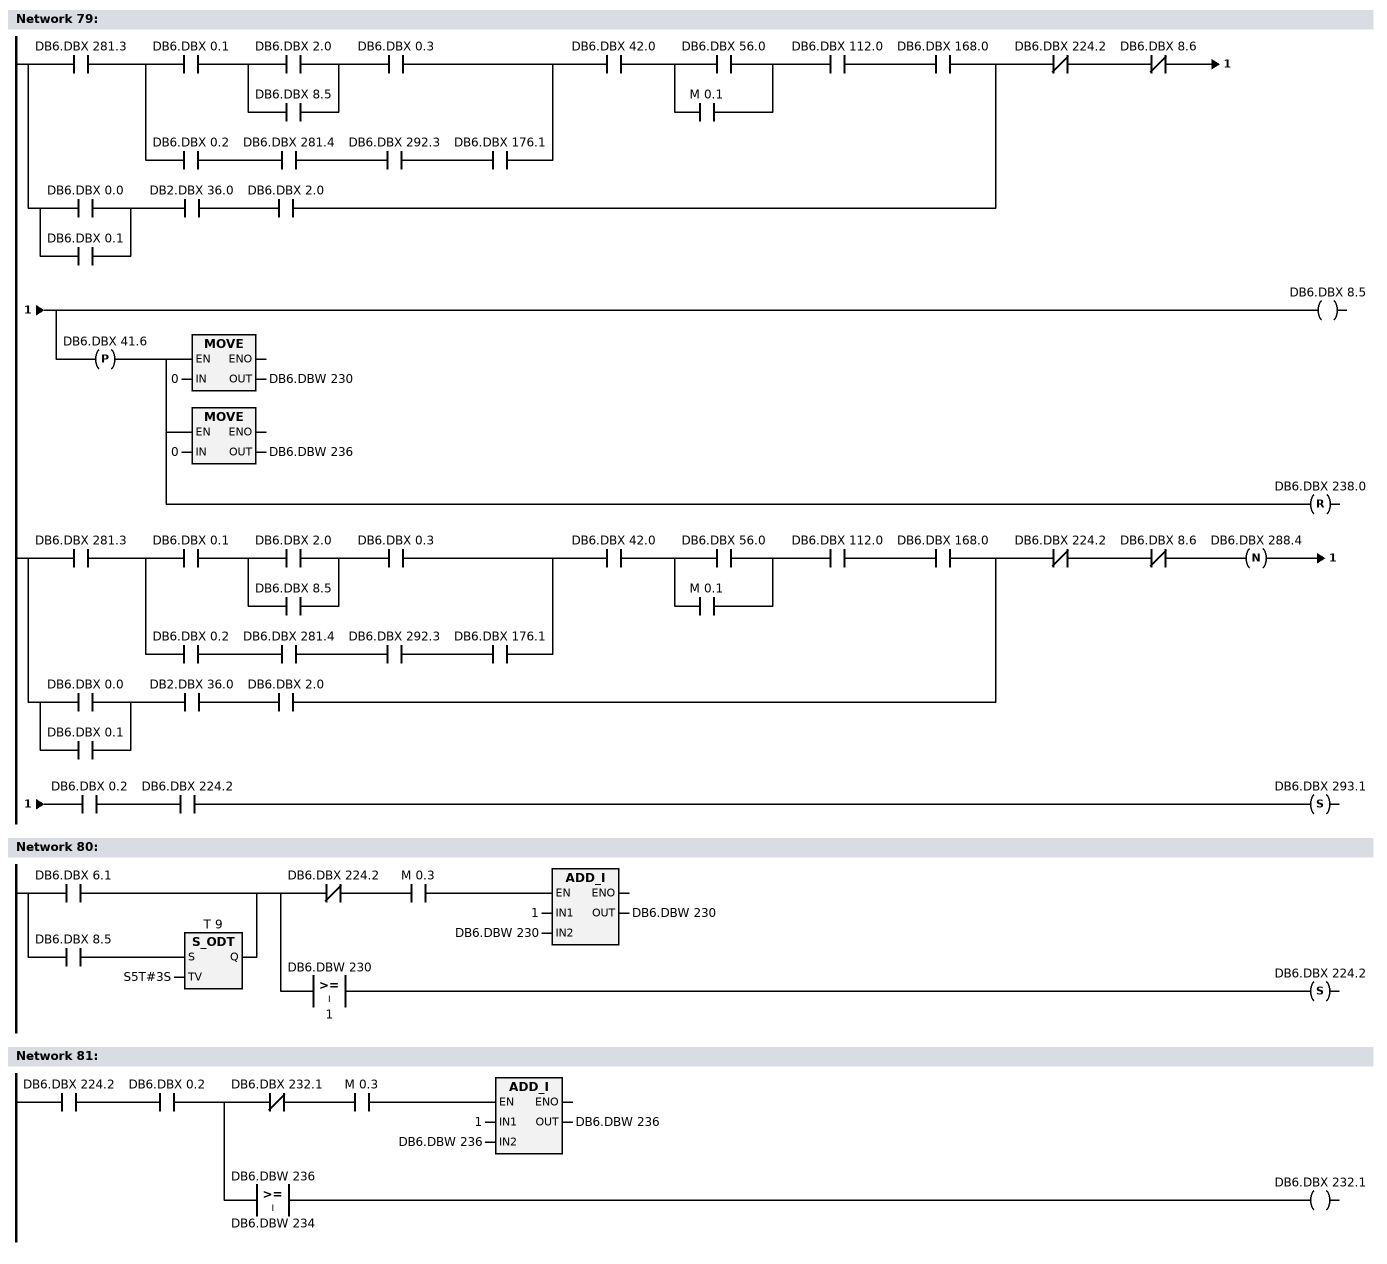
NETWORK
TITLE =
      A(;
      A     DB6.DBX 281.3;
      A(;
      A     DB6.DBX 0.1;
      A(;
      O     DB6.DBX 2.0;
      O     DB6.DBX 8.5;
      );
      A     DB6.DBX 0.3;
      O;
      A     DB6.DBX 0.2;
      A     DB6.DBX 281.4;
      A     DB6.DBX 292.3;
      A     DB6.DBX 176.1;
      );
      A     DB6.DBX 42.0;
      A(;
      O     DB6.DBX 56.0;
      O     M 0.1;
      );
      A     DB6.DBX 112.0;
      A     DB6.DBX 168.0;
      O;
      A(;
      O     DB6.DBX 0.0;
      O     DB6.DBX 0.1;
      );
      A     DB2.DBX 36.0;
      A     DB6.DBX 2.0;
      );
      AN    DB6.DBX 224.2;
      AN    DB6.DBX 8.6;
      =     L 0.0;
      A     L 0.0;
      BLD   102;
      =     DB6.DBX 8.5;
      A(;
      A     L 0.0;
      FN    DB6.DBX 288.4;
      );
      A     DB6.DBX 0.2;
      A     DB6.DBX 224.2;
      S     DB6.DBX 293.1;
      A     L 0.0;
      FP    DB6.DBX 41.6;
      =     L 0.1;
      A     L 0.1;
      JNB   M071;
      L     0;
      T     DB6.DBW 230;
M071: NOP   0;
      A     L 0.1;
      JNB   M072;
      L     0;
      T     DB6.DBW 236;
M072: NOP   0;
      A     L 0.1;
      BLD   102;
      R     DB6.DBX 238.0;
NETWORK
TITLE =
      O     DB6.DBX 6.1;
      O(;
      A     DB6.DBX 8.5;
      L     S5T#3S;
      SD    T 9;
      NOP   0;
      NOP   0;
      NOP   0;
      A     T 9;
      );
      =     L 0.0;
      A     L 0.0;
      AN    DB6.DBX 224.2;
      A     M 0.3;
      JNB   M073;
      L     1;
      L     DB6.DBW 230;
      +I;
      T     DB6.DBW 230;
M073: NOP   0;
      A     L 0.0;
      A(;
      L     DB6.DBW 230;
      L     1;
      >=I;
      );
      S     DB6.DBX 224.2;
NETWORK
TITLE =
      A     DB6.DBX 224.2;
      A     DB6.DBX 0.2;
      =     L 0.0;
      A     L 0.0;
      AN    DB6.DBX 232.1;
      A     M 0.3;
      JNB   M074;
      L     1;
      L     DB6.DBW 236;
      +I;
      T     DB6.DBW 236;
M074: NOP   0;
      A     L 0.0;
      A(;
      L     DB6.DBW 236;
      L     DB6.DBW 234;
      >=I;
      );
      =     DB6.DBX 232.1;
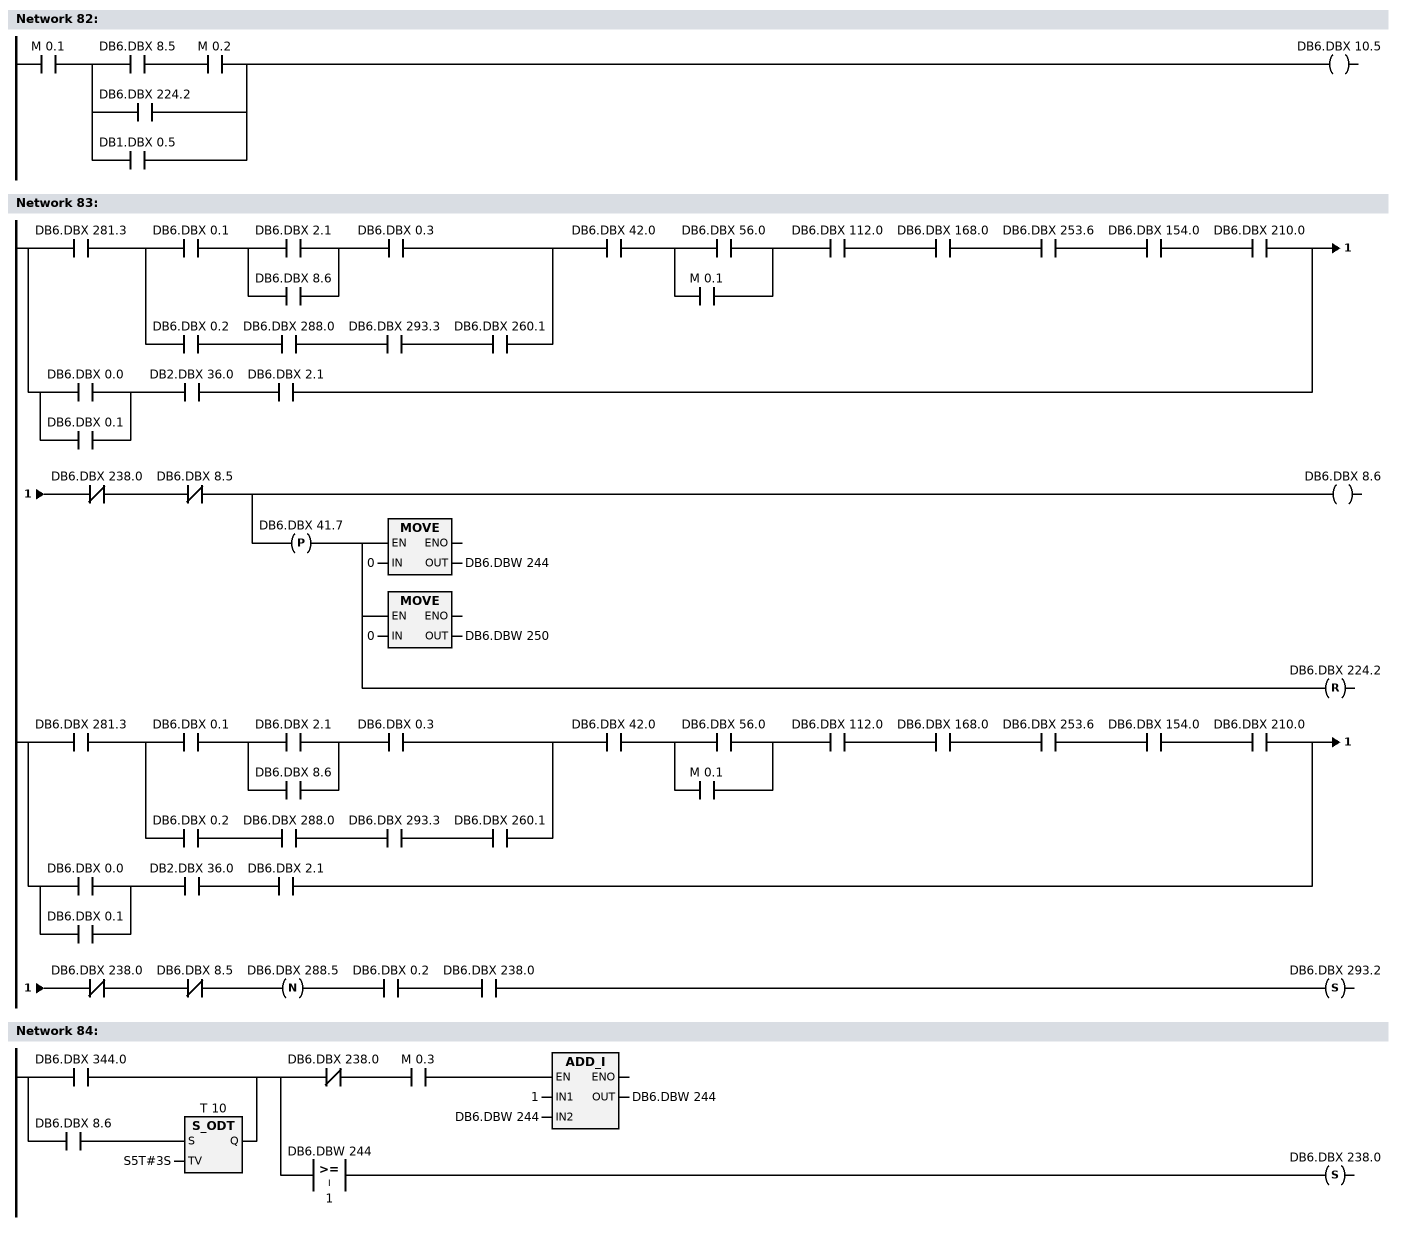
NETWORK
TITLE =
      A     M 0.1;
      A(;
      A     DB6.DBX 8.5;
      A     M 0.2;
      O     DB6.DBX 224.2;
      O     DB1.DBX 0.5;
      );
      =     DB6.DBX 10.5;
NETWORK
TITLE =
      A(;
      A     DB6.DBX 281.3;
      A(;
      A     DB6.DBX 0.1;
      A(;
      O     DB6.DBX 2.1;
      O     DB6.DBX 8.6;
      );
      A     DB6.DBX 0.3;
      O;
      A     DB6.DBX 0.2;
      A     DB6.DBX 288.0;
      A     DB6.DBX 293.3;
      A     DB6.DBX 260.1;
      );
      A     DB6.DBX 42.0;
      A(;
      O     DB6.DBX 56.0;
      O     M 0.1;
      );
      A     DB6.DBX 112.0;
      A     DB6.DBX 168.0;
      A     DB6.DBX 253.6;
      A     DB6.DBX 154.0;
      A     DB6.DBX 210.0;
      O;
      A(;
      O     DB6.DBX 0.0;
      O     DB6.DBX 0.1;
      );
      A     DB2.DBX 36.0;
      A     DB6.DBX 2.1;
      );
      AN    DB6.DBX 238.0;
      AN    DB6.DBX 8.5;
      =     L 0.0;
      A     L 0.0;
      BLD   102;
      =     DB6.DBX 8.6;
      A(;
      A     L 0.0;
      FN    DB6.DBX 288.5;
      );
      A     DB6.DBX 0.2;
      A     DB6.DBX 238.0;
      S     DB6.DBX 293.2;
      A     L 0.0;
      FP    DB6.DBX 41.7;
      =     L 0.1;
      A     L 0.1;
      JNB   M075;
      L     0;
      T     DB6.DBW 244;
M075: NOP   0;
      A     L 0.1;
      JNB   M076;
      L     0;
      T     DB6.DBW 250;
M076: NOP   0;
      A     L 0.1;
      BLD   102;
      R     DB6.DBX 224.2;
NETWORK
TITLE =
      O     DB6.DBX 344.0;
      O(;
      A     DB6.DBX 8.6;
      L     S5T#3S;
      SD    T 10;
      NOP   0;
      NOP   0;
      NOP   0;
      A     T 10;
      );
      =     L 0.0;
      A     L 0.0;
      AN    DB6.DBX 238.0;
      A     M 0.3;
      JNB   M077;
      L     1;
      L     DB6.DBW 244;
      +I;
      T     DB6.DBW 244;
M077: NOP   0;
      A     L 0.0;
      A(;
      L     DB6.DBW 244;
      L     1;
      >=I;
      );
      S     DB6.DBX 238.0;
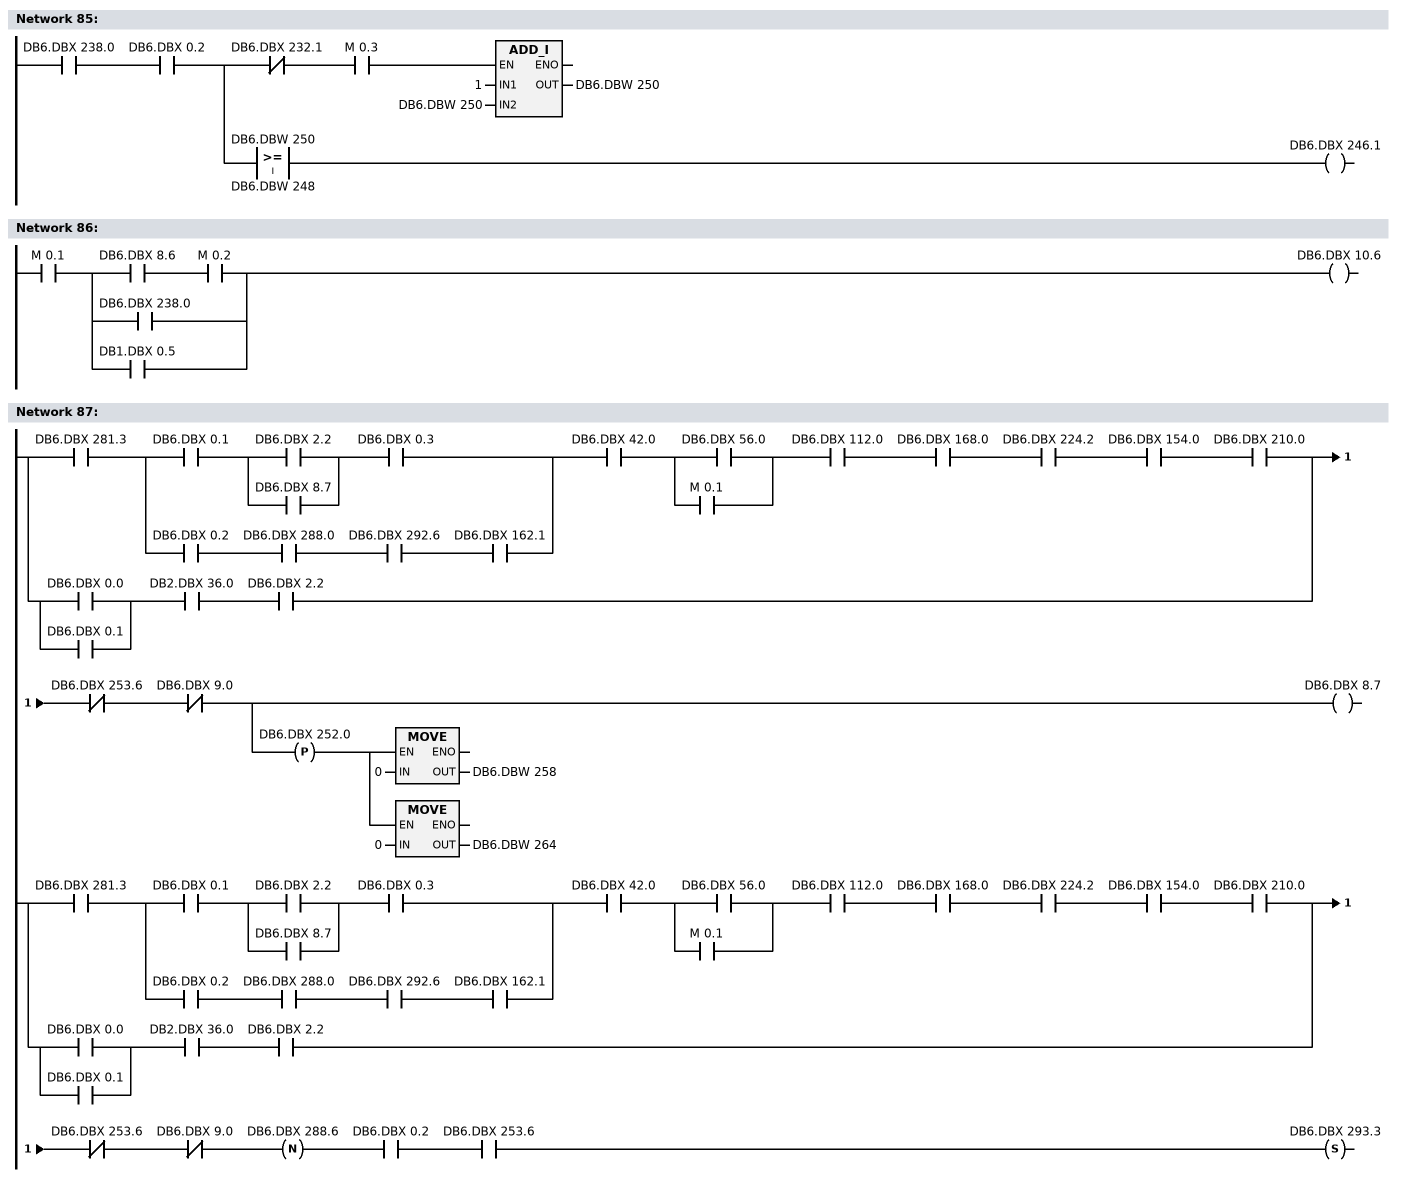
NETWORK
TITLE =
      A     DB6.DBX 238.0;
      A     DB6.DBX 0.2;
      =     L 0.0;
      A     L 0.0;
      AN    DB6.DBX 232.1;
      A     M 0.3;
      JNB   M078;
      L     1;
      L     DB6.DBW 250;
      +I;
      T     DB6.DBW 250;
M078: NOP   0;
      A     L 0.0;
      A(;
      L     DB6.DBW 250;
      L     DB6.DBW 248;
      >=I;
      );
      =     DB6.DBX 246.1;
NETWORK
TITLE =
      A     M 0.1;
      A(;
      A     DB6.DBX 8.6;
      A     M 0.2;
      O     DB6.DBX 238.0;
      O     DB1.DBX 0.5;
      );
      =     DB6.DBX 10.6;
NETWORK
TITLE =
      A(;
      A     DB6.DBX 281.3;
      A(;
      A     DB6.DBX 0.1;
      A(;
      O     DB6.DBX 2.2;
      O     DB6.DBX 8.7;
      );
      A     DB6.DBX 0.3;
      O;
      A     DB6.DBX 0.2;
      A     DB6.DBX 288.0;
      A     DB6.DBX 292.6;
      A     DB6.DBX 162.1;
      );
      A     DB6.DBX 42.0;
      A(;
      O     DB6.DBX 56.0;
      O     M 0.1;
      );
      A     DB6.DBX 112.0;
      A     DB6.DBX 168.0;
      A     DB6.DBX 224.2;
      A     DB6.DBX 154.0;
      A     DB6.DBX 210.0;
      O;
      A(;
      O     DB6.DBX 0.0;
      O     DB6.DBX 0.1;
      );
      A     DB2.DBX 36.0;
      A     DB6.DBX 2.2;
      );
      AN    DB6.DBX 253.6;
      AN    DB6.DBX 9.0;
      =     L 0.0;
      A     L 0.0;
      BLD   102;
      =     DB6.DBX 8.7;
      A(;
      A     L 0.0;
      FN    DB6.DBX 288.6;
      );
      A     DB6.DBX 0.2;
      A     DB6.DBX 253.6;
      S     DB6.DBX 293.3;
      A     L 0.0;
      FP    DB6.DBX 252.0;
      =     L 0.1;
      A     L 0.1;
      JNB   M079;
      L     0;
      T     DB6.DBW 258;
M079: NOP   0;
      A     L 0.1;
      JNB   M080;
      L     0;
      T     DB6.DBW 264;
M080: NOP   0;
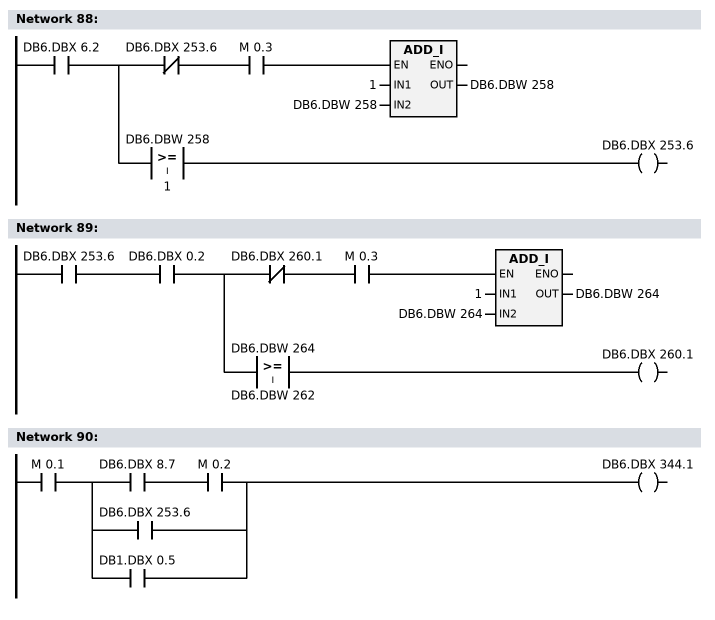
NETWORK
TITLE =
      A     DB6.DBX 6.2;
      =     L 0.0;
      A     L 0.0;
      AN    DB6.DBX 253.6;
      A     M 0.3;
      JNB   M081;
      L     1;
      L     DB6.DBW 258;
      +I;
      T     DB6.DBW 258;
M081: NOP   0;
      A     L 0.0;
      A(;
      L     DB6.DBW 258;
      L     1;
      >=I;
      );
      =     DB6.DBX 253.6;
NETWORK
TITLE =
      A     DB6.DBX 253.6;
      A     DB6.DBX 0.2;
      =     L 0.0;
      A     L 0.0;
      AN    DB6.DBX 260.1;
      A     M 0.3;
      JNB   M082;
      L     1;
      L     DB6.DBW 264;
      +I;
      T     DB6.DBW 264;
M082: NOP   0;
      A     L 0.0;
      A(;
      L     DB6.DBW 264;
      L     DB6.DBW 262;
      >=I;
      );
      =     DB6.DBX 260.1;
NETWORK
TITLE =
      A     M 0.1;
      A(;
      A     DB6.DBX 8.7;
      A     M 0.2;
      O     DB6.DBX 253.6;
      O     DB1.DBX 0.5;
      );
      =     DB6.DBX 344.1;
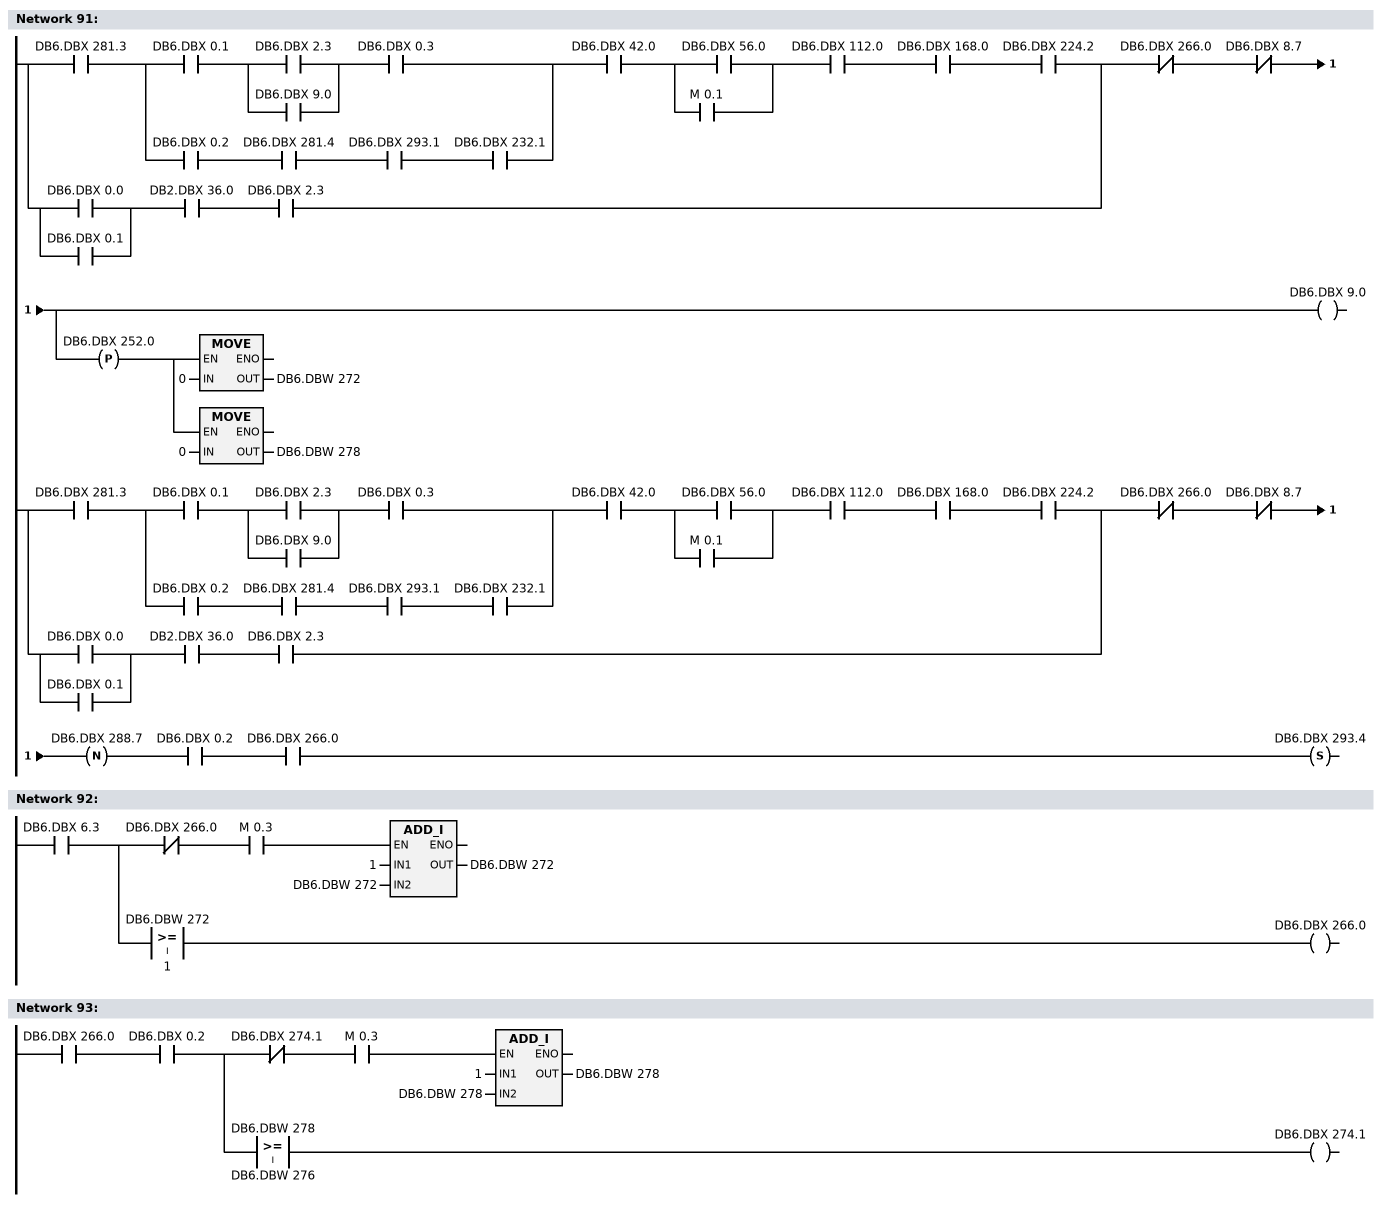
NETWORK
TITLE =
      A(;
      A     DB6.DBX 281.3;
      A(;
      A     DB6.DBX 0.1;
      A(;
      O     DB6.DBX 2.3;
      O     DB6.DBX 9.0;
      );
      A     DB6.DBX 0.3;
      O;
      A     DB6.DBX 0.2;
      A     DB6.DBX 281.4;
      A     DB6.DBX 293.1;
      A     DB6.DBX 232.1;
      );
      A     DB6.DBX 42.0;
      A(;
      O     DB6.DBX 56.0;
      O     M 0.1;
      );
      A     DB6.DBX 112.0;
      A     DB6.DBX 168.0;
      A     DB6.DBX 224.2;
      O;
      A(;
      O     DB6.DBX 0.0;
      O     DB6.DBX 0.1;
      );
      A     DB2.DBX 36.0;
      A     DB6.DBX 2.3;
      );
      AN    DB6.DBX 266.0;
      AN    DB6.DBX 8.7;
      =     L 0.0;
      A     L 0.0;
      BLD   102;
      =     DB6.DBX 9.0;
      A(;
      A     L 0.0;
      FN    DB6.DBX 288.7;
      );
      A     DB6.DBX 0.2;
      A     DB6.DBX 266.0;
      S     DB6.DBX 293.4;
      A     L 0.0;
      FP    DB6.DBX 252.0;
      =     L 0.1;
      A     L 0.1;
      JNB   M083;
      L     0;
      T     DB6.DBW 272;
M083: NOP   0;
      A     L 0.1;
      JNB   M084;
      L     0;
      T     DB6.DBW 278;
M084: NOP   0;
NETWORK
TITLE =
      A     DB6.DBX 6.3;
      =     L 0.0;
      A     L 0.0;
      AN    DB6.DBX 266.0;
      A     M 0.3;
      JNB   M085;
      L     1;
      L     DB6.DBW 272;
      +I;
      T     DB6.DBW 272;
M085: NOP   0;
      A     L 0.0;
      A(;
      L     DB6.DBW 272;
      L     1;
      >=I;
      );
      =     DB6.DBX 266.0;
NETWORK
TITLE =
      A     DB6.DBX 266.0;
      A     DB6.DBX 0.2;
      =     L 0.0;
      A     L 0.0;
      AN    DB6.DBX 274.1;
      A     M 0.3;
      JNB   M086;
      L     1;
      L     DB6.DBW 278;
      +I;
      T     DB6.DBW 278;
M086: NOP   0;
      A     L 0.0;
      A(;
      L     DB6.DBW 278;
      L     DB6.DBW 276;
      >=I;
      );
      =     DB6.DBX 274.1;
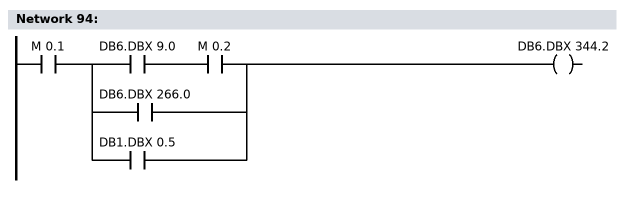
NETWORK
TITLE =
      A     M 0.1;
      A(;
      A     DB6.DBX 9.0;
      A     M 0.2;
      O     DB6.DBX 266.0;
      O     DB1.DBX 0.5;
      );
      =     DB6.DBX 344.2;
END_FUNCTION

FUNCTION FC 9 : VOID
AUTHOR : Kamillas
VERSION : 0.1
BEGIN
// (block stored without names or comments; labels and parameter names are numbered)
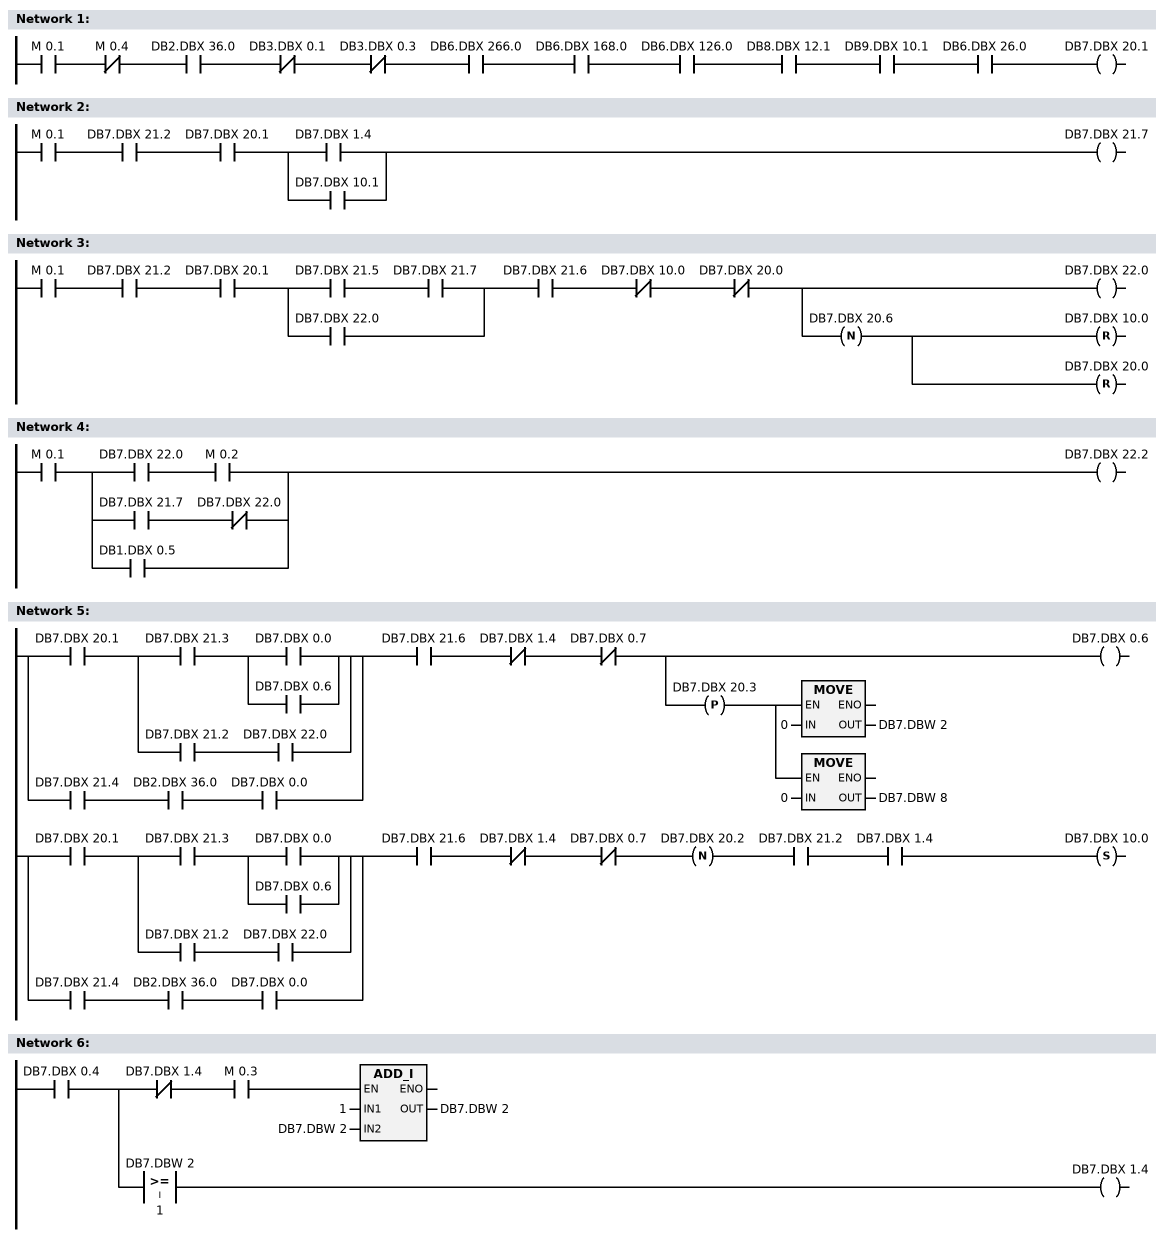
NETWORK
TITLE =
      A     M 0.1;
      AN    M 0.4;
      A     DB2.DBX 36.0;
      AN    DB3.DBX 0.1;
      AN    DB3.DBX 0.3;
      A     DB6.DBX 266.0;
      A     DB6.DBX 168.0;
      A     DB6.DBX 126.0;
      A     DB8.DBX 12.1;
      A     DB9.DBX 10.1;
      A     DB6.DBX 26.0;
      =     DB7.DBX 20.1;
NETWORK
TITLE =
      A     M 0.1;
      A     DB7.DBX 21.2;
      A     DB7.DBX 20.1;
      A(;
      O     DB7.DBX 1.4;
      O     DB7.DBX 10.1;
      );
      =     DB7.DBX 21.7;
NETWORK
TITLE =
      A     M 0.1;
      A     DB7.DBX 21.2;
      A     DB7.DBX 20.1;
      A(;
      A     DB7.DBX 21.5;
      A     DB7.DBX 21.7;
      O     DB7.DBX 22.0;
      );
      A     DB7.DBX 21.6;
      AN    DB7.DBX 10.0;
      AN    DB7.DBX 20.0;
      =     L 0.0;
      A     L 0.0;
      BLD   102;
      =     DB7.DBX 22.0;
      A     L 0.0;
      FN    DB7.DBX 20.6;
      R     DB7.DBX 10.0;
      R     DB7.DBX 20.0;
NETWORK
TITLE =
      A     M 0.1;
      A(;
      A     DB7.DBX 22.0;
      A     M 0.2;
      O;
      A     DB7.DBX 21.7;
      AN    DB7.DBX 22.0;
      O     DB1.DBX 0.5;
      );
      =     DB7.DBX 22.2;
NETWORK
TITLE =
      A(;
      A     DB7.DBX 20.1;
      A(;
      A     DB7.DBX 21.3;
      A(;
      O     DB7.DBX 0.0;
      O     DB7.DBX 0.6;
      );
      O;
      A     DB7.DBX 21.2;
      A     DB7.DBX 22.0;
      );
      O;
      A     DB7.DBX 21.4;
      A     DB2.DBX 36.0;
      A     DB7.DBX 0.0;
      );
      A     DB7.DBX 21.6;
      AN    DB7.DBX 1.4;
      AN    DB7.DBX 0.7;
      =     L 0.0;
      A     L 0.0;
      BLD   102;
      =     DB7.DBX 0.6;
      A(;
      A     L 0.0;
      FN    DB7.DBX 20.2;
      );
      A     DB7.DBX 21.2;
      A     DB7.DBX 1.4;
      S     DB7.DBX 10.0;
      A     L 0.0;
      FP    DB7.DBX 20.3;
      =     L 0.1;
      A     L 0.1;
      JNB   M001;
      L     0;
      T     DB7.DBW 2;
M001: NOP   0;
      A     L 0.1;
      JNB   M002;
      L     0;
      T     DB7.DBW 8;
M002: NOP   0;
NETWORK
TITLE =
      A     DB7.DBX 0.4;
      =     L 0.0;
      A     L 0.0;
      AN    DB7.DBX 1.4;
      A     M 0.3;
      JNB   M003;
      L     1;
      L     DB7.DBW 2;
      +I;
      T     DB7.DBW 2;
M003: NOP   0;
      A     L 0.0;
      A(;
      L     DB7.DBW 2;
      L     1;
      >=I;
      );
      =     DB7.DBX 1.4;
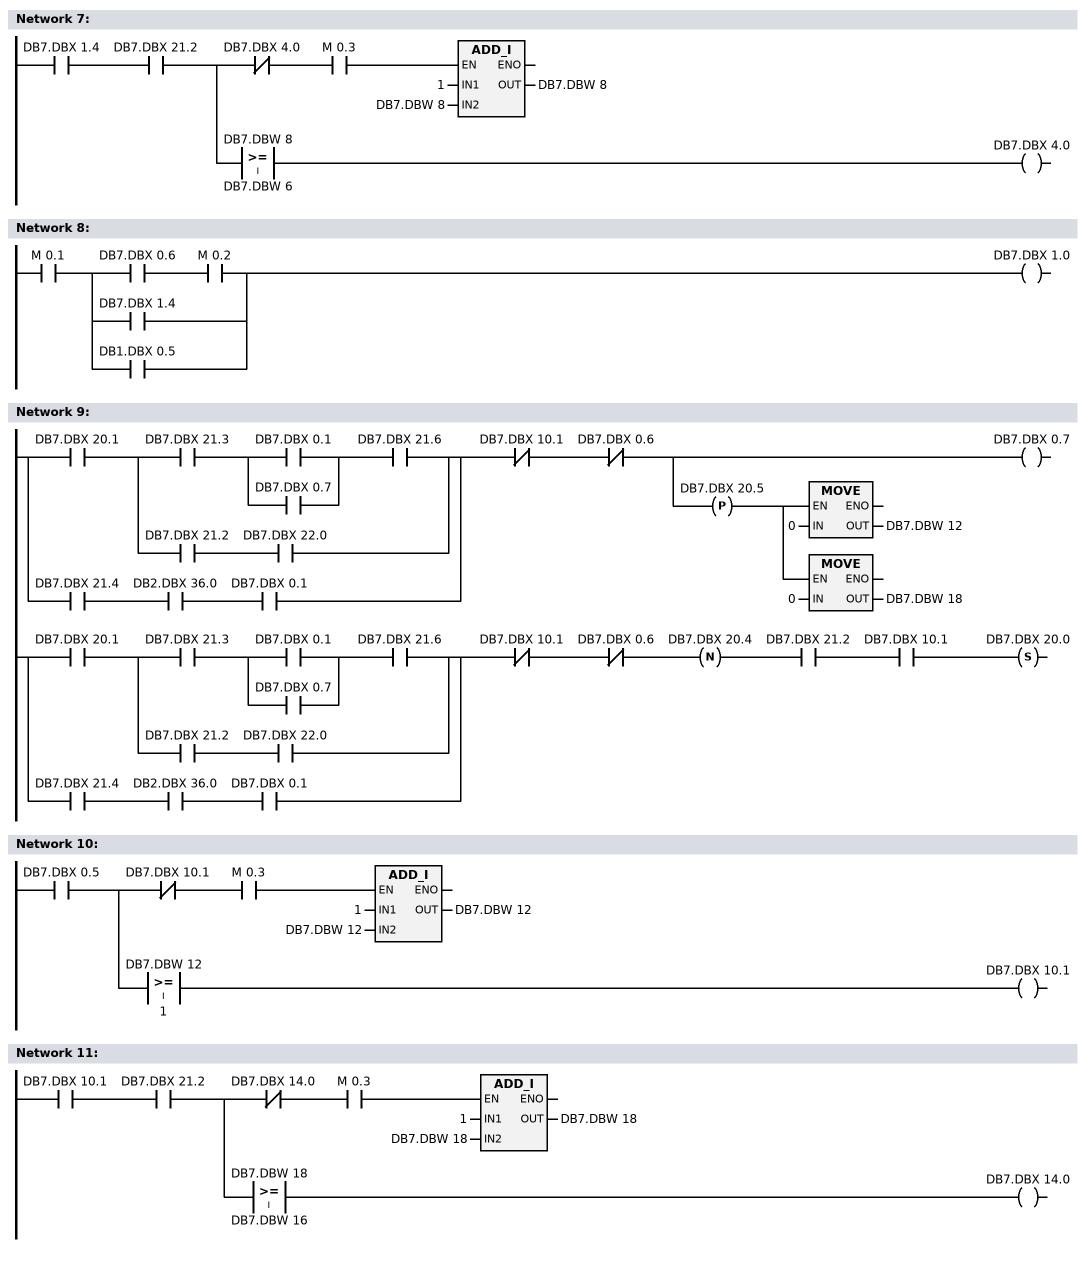
NETWORK
TITLE =
      A     DB7.DBX 1.4;
      A     DB7.DBX 21.2;
      =     L 0.0;
      A     L 0.0;
      AN    DB7.DBX 4.0;
      A     M 0.3;
      JNB   M004;
      L     1;
      L     DB7.DBW 8;
      +I;
      T     DB7.DBW 8;
M004: NOP   0;
      A     L 0.0;
      A(;
      L     DB7.DBW 8;
      L     DB7.DBW 6;
      >=I;
      );
      =     DB7.DBX 4.0;
NETWORK
TITLE =
      A     M 0.1;
      A(;
      A     DB7.DBX 0.6;
      A     M 0.2;
      O     DB7.DBX 1.4;
      O     DB1.DBX 0.5;
      );
      =     DB7.DBX 1.0;
NETWORK
TITLE =
      A(;
      A     DB7.DBX 20.1;
      A(;
      A     DB7.DBX 21.3;
      A(;
      O     DB7.DBX 0.1;
      O     DB7.DBX 0.7;
      );
      A     DB7.DBX 21.6;
      O;
      A     DB7.DBX 21.2;
      A     DB7.DBX 22.0;
      );
      O;
      A     DB7.DBX 21.4;
      A     DB2.DBX 36.0;
      A     DB7.DBX 0.1;
      );
      AN    DB7.DBX 10.1;
      AN    DB7.DBX 0.6;
      =     L 0.0;
      A     L 0.0;
      BLD   102;
      =     DB7.DBX 0.7;
      A(;
      A     L 0.0;
      FN    DB7.DBX 20.4;
      );
      A     DB7.DBX 21.2;
      A     DB7.DBX 10.1;
      S     DB7.DBX 20.0;
      A     L 0.0;
      FP    DB7.DBX 20.5;
      =     L 0.1;
      A     L 0.1;
      JNB   M005;
      L     0;
      T     DB7.DBW 12;
M005: NOP   0;
      A     L 0.1;
      JNB   M006;
      L     0;
      T     DB7.DBW 18;
M006: NOP   0;
NETWORK
TITLE =
      A     DB7.DBX 0.5;
      =     L 0.0;
      A     L 0.0;
      AN    DB7.DBX 10.1;
      A     M 0.3;
      JNB   M007;
      L     1;
      L     DB7.DBW 12;
      +I;
      T     DB7.DBW 12;
M007: NOP   0;
      A     L 0.0;
      A(;
      L     DB7.DBW 12;
      L     1;
      >=I;
      );
      =     DB7.DBX 10.1;
NETWORK
TITLE =
      A     DB7.DBX 10.1;
      A     DB7.DBX 21.2;
      =     L 0.0;
      A     L 0.0;
      AN    DB7.DBX 14.0;
      A     M 0.3;
      JNB   M008;
      L     1;
      L     DB7.DBW 18;
      +I;
      T     DB7.DBW 18;
M008: NOP   0;
      A     L 0.0;
      A(;
      L     DB7.DBW 18;
      L     DB7.DBW 16;
      >=I;
      );
      =     DB7.DBX 14.0;
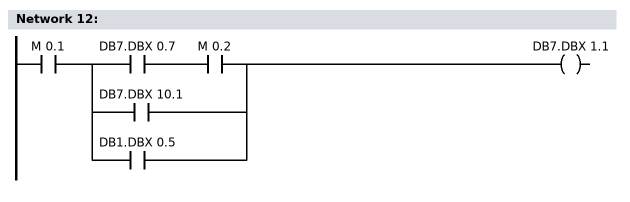
NETWORK
TITLE =
      A     M 0.1;
      A(;
      A     DB7.DBX 0.7;
      A     M 0.2;
      O     DB7.DBX 10.1;
      O     DB1.DBX 0.5;
      );
      =     DB7.DBX 1.1;
END_FUNCTION

FUNCTION FC 10 : VOID
AUTHOR : Kamillas
VERSION : 0.1
BEGIN
// (block stored without names or comments; labels and parameter names are numbered)
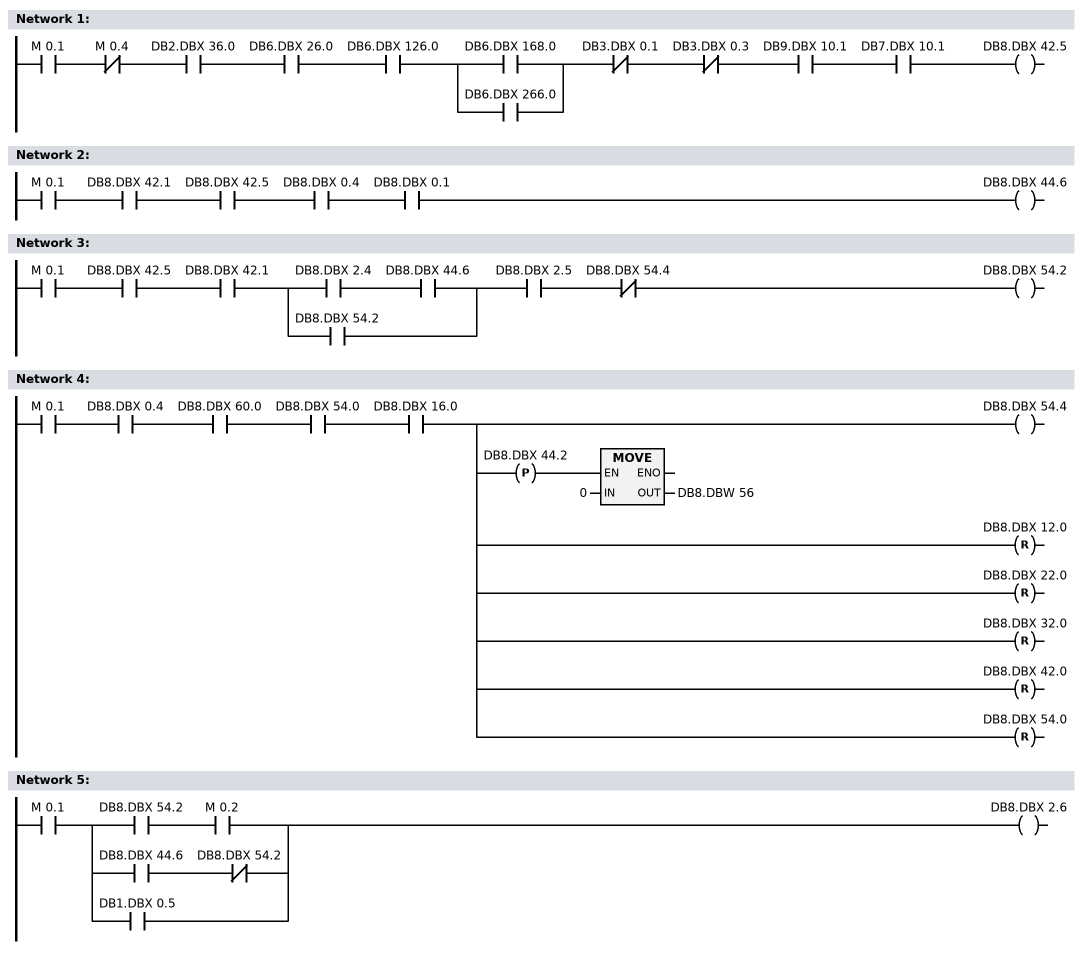
NETWORK
TITLE =
      A     M 0.1;
      AN    M 0.4;
      A     DB2.DBX 36.0;
      A     DB6.DBX 26.0;
      A     DB6.DBX 126.0;
      A(;
      O     DB6.DBX 168.0;
      O     DB6.DBX 266.0;
      );
      AN    DB3.DBX 0.1;
      AN    DB3.DBX 0.3;
      A     DB9.DBX 10.1;
      A     DB7.DBX 10.1;
      =     DB8.DBX 42.5;
NETWORK
TITLE =
      A     M 0.1;
      A     DB8.DBX 42.1;
      A     DB8.DBX 42.5;
      A     DB8.DBX 0.4;
      A     DB8.DBX 0.1;
      =     DB8.DBX 44.6;
NETWORK
TITLE =
      A     M 0.1;
      A     DB8.DBX 42.5;
      A     DB8.DBX 42.1;
      A(;
      A     DB8.DBX 2.4;
      A     DB8.DBX 44.6;
      O     DB8.DBX 54.2;
      );
      A     DB8.DBX 2.5;
      AN    DB8.DBX 54.4;
      =     DB8.DBX 54.2;
NETWORK
TITLE =
      A     M 0.1;
      A     DB8.DBX 0.4;
      A     DB8.DBX 60.0;
      A     DB8.DBX 54.0;
      A     DB8.DBX 16.0;
      =     L 0.0;
      A     L 0.0;
      BLD   102;
      =     DB8.DBX 54.4;
      A     L 0.0;
      FP    DB8.DBX 44.2;
      JNB   M001;
      L     0;
      T     DB8.DBW 56;
M001: NOP   0;
      A     L 0.0;
      BLD   102;
      R     DB8.DBX 12.0;
      A     L 0.0;
      BLD   102;
      R     DB8.DBX 22.0;
      A     L 0.0;
      BLD   102;
      R     DB8.DBX 32.0;
      A     L 0.0;
      BLD   102;
      R     DB8.DBX 42.0;
      A     L 0.0;
      BLD   102;
      R     DB8.DBX 54.0;
NETWORK
TITLE =
      A     M 0.1;
      A(;
      A     DB8.DBX 54.2;
      A     M 0.2;
      O;
      A     DB8.DBX 44.6;
      AN    DB8.DBX 54.2;
      O     DB1.DBX 0.5;
      );
      =     DB8.DBX 2.6;
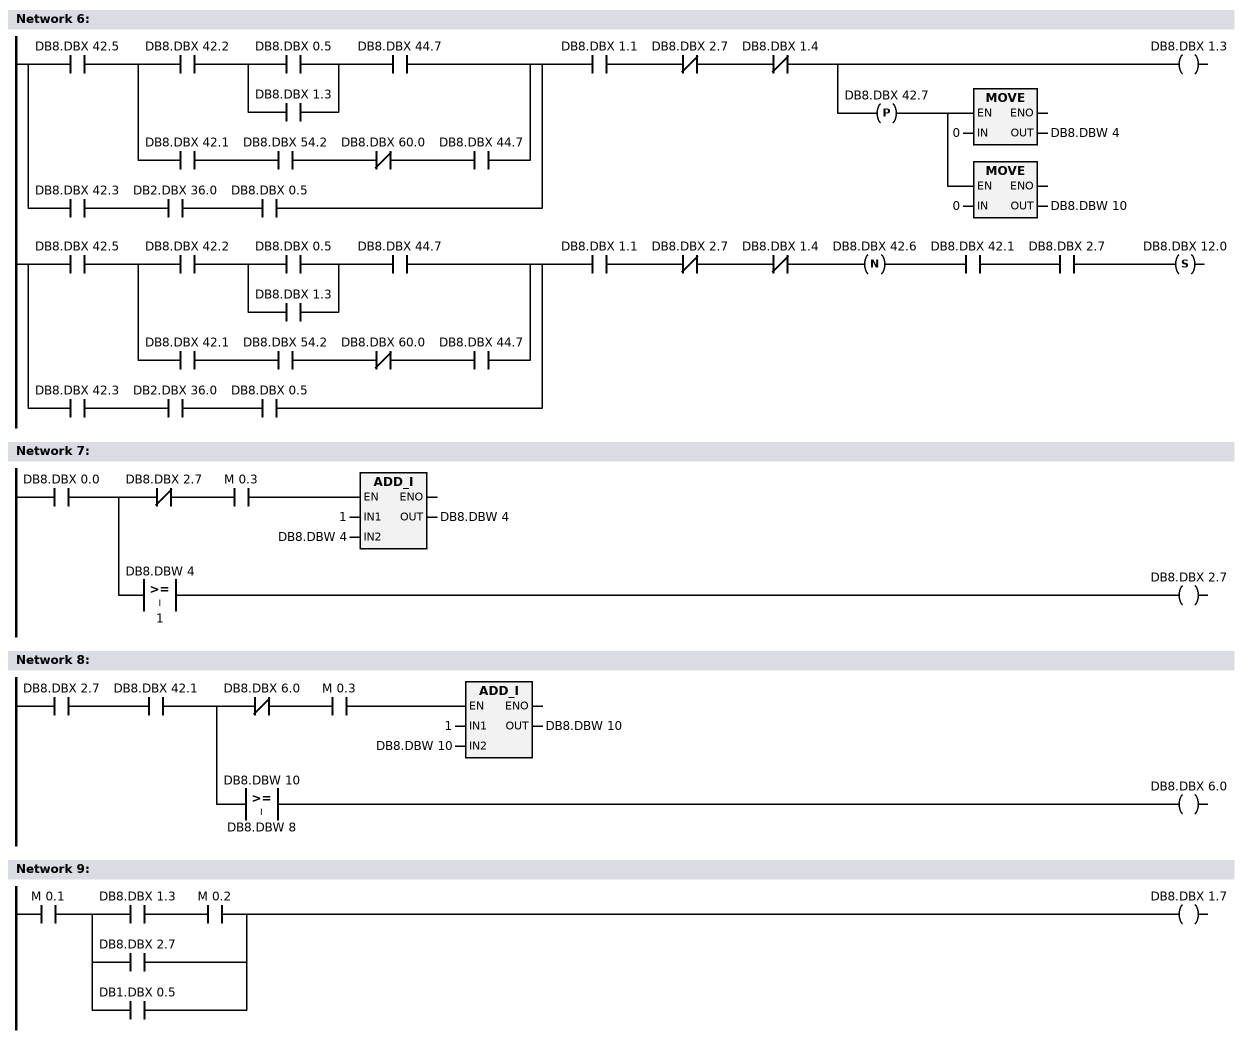
NETWORK
TITLE =
      A(;
      A     DB8.DBX 42.5;
      A(;
      A     DB8.DBX 42.2;
      A(;
      O     DB8.DBX 0.5;
      O     DB8.DBX 1.3;
      );
      A     DB8.DBX 44.7;
      O;
      A     DB8.DBX 42.1;
      A     DB8.DBX 54.2;
      AN    DB8.DBX 60.0;
      A     DB8.DBX 44.7;
      );
      O;
      A     DB8.DBX 42.3;
      A     DB2.DBX 36.0;
      A     DB8.DBX 0.5;
      );
      A     DB8.DBX 1.1;
      AN    DB8.DBX 2.7;
      AN    DB8.DBX 1.4;
      =     L 0.0;
      A     L 0.0;
      BLD   102;
      =     DB8.DBX 1.3;
      A(;
      A     L 0.0;
      FN    DB8.DBX 42.6;
      );
      A     DB8.DBX 42.1;
      A     DB8.DBX 2.7;
      S     DB8.DBX 12.0;
      A     L 0.0;
      FP    DB8.DBX 42.7;
      =     L 0.1;
      A     L 0.1;
      JNB   M002;
      L     0;
      T     DB8.DBW 4;
M002: NOP   0;
      A     L 0.1;
      JNB   M003;
      L     0;
      T     DB8.DBW 10;
M003: NOP   0;
NETWORK
TITLE =
      A     DB8.DBX 0.0;
      =     L 0.0;
      A     L 0.0;
      AN    DB8.DBX 2.7;
      A     M 0.3;
      JNB   M004;
      L     1;
      L     DB8.DBW 4;
      +I;
      T     DB8.DBW 4;
M004: NOP   0;
      A     L 0.0;
      A(;
      L     DB8.DBW 4;
      L     1;
      >=I;
      );
      =     DB8.DBX 2.7;
NETWORK
TITLE =
      A     DB8.DBX 2.7;
      A     DB8.DBX 42.1;
      =     L 0.0;
      A     L 0.0;
      AN    DB8.DBX 6.0;
      A     M 0.3;
      JNB   M005;
      L     1;
      L     DB8.DBW 10;
      +I;
      T     DB8.DBW 10;
M005: NOP   0;
      A     L 0.0;
      A(;
      L     DB8.DBW 10;
      L     DB8.DBW 8;
      >=I;
      );
      =     DB8.DBX 6.0;
NETWORK
TITLE =
      A     M 0.1;
      A(;
      A     DB8.DBX 1.3;
      A     M 0.2;
      O     DB8.DBX 2.7;
      O     DB1.DBX 0.5;
      );
      =     DB8.DBX 1.7;
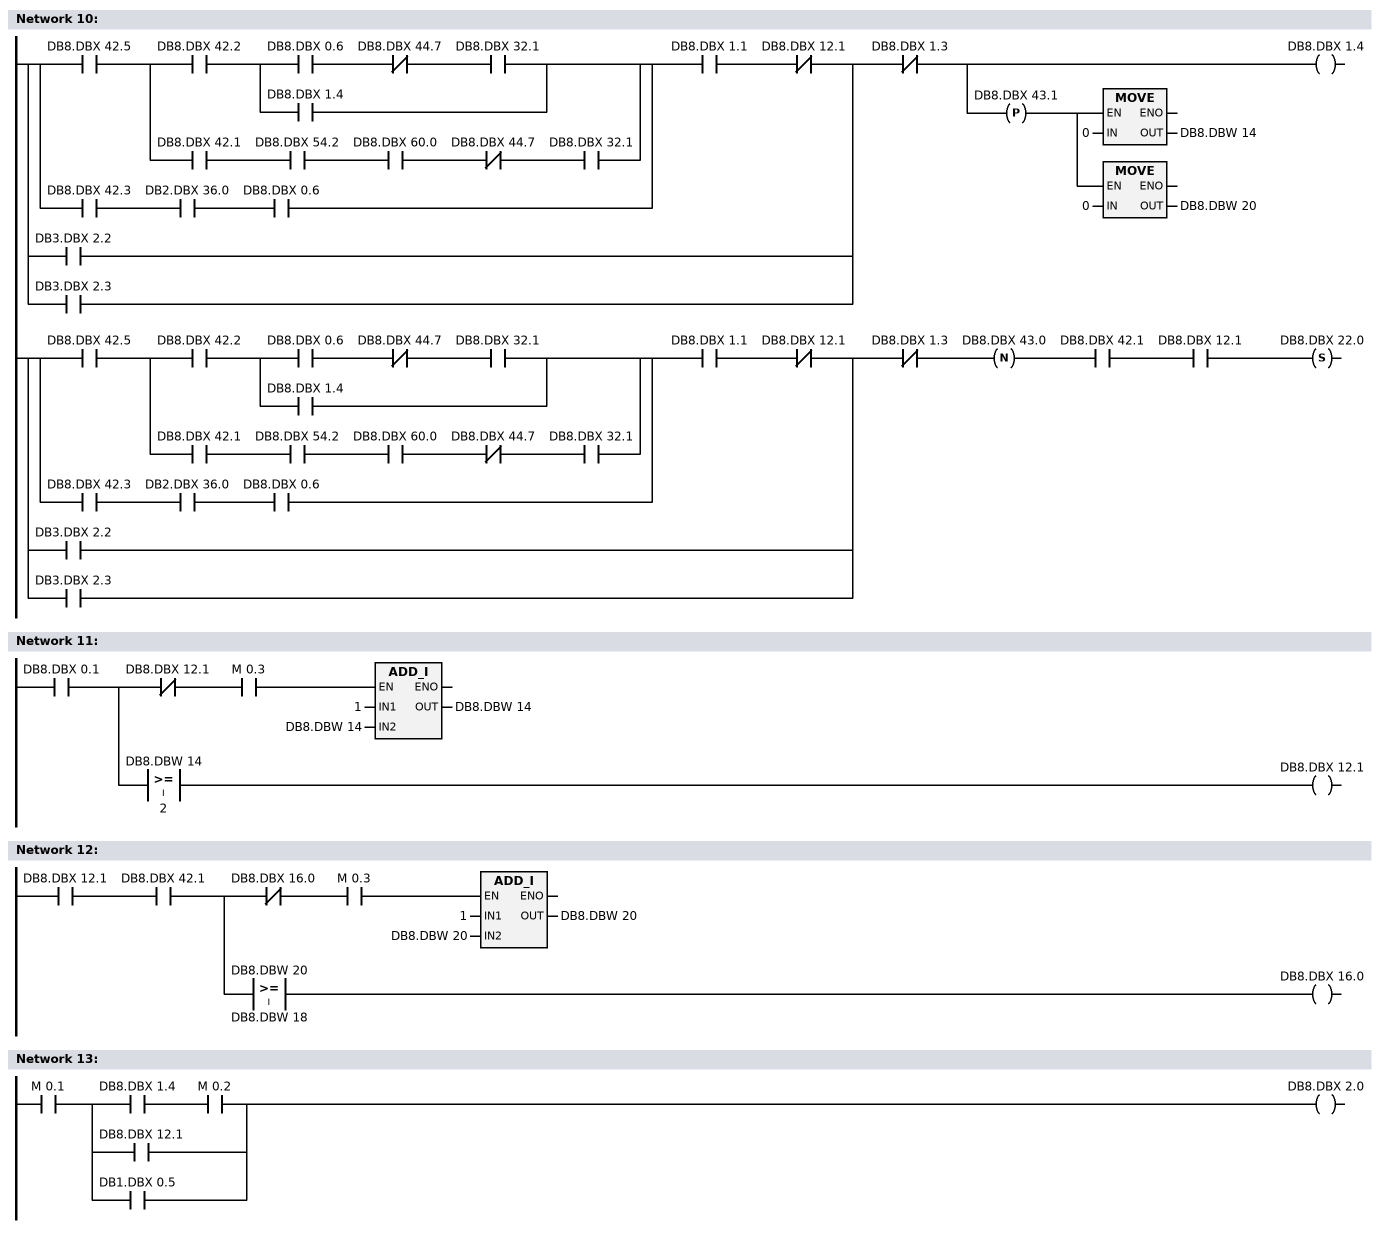
NETWORK
TITLE =
      A(;
      A(;
      A     DB8.DBX 42.5;
      A(;
      A     DB8.DBX 42.2;
      A(;
      A     DB8.DBX 0.6;
      AN    DB8.DBX 44.7;
      A     DB8.DBX 32.1;
      O     DB8.DBX 1.4;
      );
      O;
      A     DB8.DBX 42.1;
      A     DB8.DBX 54.2;
      A     DB8.DBX 60.0;
      AN    DB8.DBX 44.7;
      A     DB8.DBX 32.1;
      );
      O;
      A     DB8.DBX 42.3;
      A     DB2.DBX 36.0;
      A     DB8.DBX 0.6;
      );
      A     DB8.DBX 1.1;
      AN    DB8.DBX 12.1;
      O     DB3.DBX 2.2;
      O     DB3.DBX 2.3;
      );
      AN    DB8.DBX 1.3;
      =     L 0.0;
      A     L 0.0;
      BLD   102;
      =     DB8.DBX 1.4;
      A(;
      A     L 0.0;
      FN    DB8.DBX 43.0;
      );
      A     DB8.DBX 42.1;
      A     DB8.DBX 12.1;
      S     DB8.DBX 22.0;
      A     L 0.0;
      FP    DB8.DBX 43.1;
      =     L 0.1;
      A     L 0.1;
      JNB   M006;
      L     0;
      T     DB8.DBW 14;
M006: NOP   0;
      A     L 0.1;
      JNB   M007;
      L     0;
      T     DB8.DBW 20;
M007: NOP   0;
NETWORK
TITLE =
      A     DB8.DBX 0.1;
      =     L 0.0;
      A     L 0.0;
      AN    DB8.DBX 12.1;
      A     M 0.3;
      JNB   M008;
      L     1;
      L     DB8.DBW 14;
      +I;
      T     DB8.DBW 14;
M008: NOP   0;
      A     L 0.0;
      A(;
      L     DB8.DBW 14;
      L     2;
      >=I;
      );
      =     DB8.DBX 12.1;
NETWORK
TITLE =
      A     DB8.DBX 12.1;
      A     DB8.DBX 42.1;
      =     L 0.0;
      A     L 0.0;
      AN    DB8.DBX 16.0;
      A     M 0.3;
      JNB   M009;
      L     1;
      L     DB8.DBW 20;
      +I;
      T     DB8.DBW 20;
M009: NOP   0;
      A     L 0.0;
      A(;
      L     DB8.DBW 20;
      L     DB8.DBW 18;
      >=I;
      );
      =     DB8.DBX 16.0;
NETWORK
TITLE =
      A     M 0.1;
      A(;
      A     DB8.DBX 1.4;
      A     M 0.2;
      O     DB8.DBX 12.1;
      O     DB1.DBX 0.5;
      );
      =     DB8.DBX 2.0;
